// TIA Portal V20 export
FUNCTION_BLOCK "zPMC_Map"   // FB77, LAD
// stored: MemoryReserve 100, Namespace CITI_Logic, SetENOAutomatically false
   VAR_INPUT
      IN_AssistanceCall : Array[1..8] of Bool;
      IN_AssistanceCallAck : Array[1..8] of Bool;
      IN_Configuration : "CITI_Logic.zp_CITI_Configuration";
      IN_Data : "CITI_Logic.PMC_Input_Data";
   END_VAR
   VAR_OUTPUT
      OUT_Flasher_1Hz : Bool;   // 1Hz Flashing bit
      OUT_Team_Leader_Call_Out : Bool;   // ON when a Team Leader Call is active
      OUT_ShiftNumber : Byte;
   END_VAR
   VAR_IN_OUT
      PMC_Data : "CITI_Logic.zp_CITIData";
   END_VAR
   VAR
      MM_FaultWord_Zero : Bool;
      CycleTime_RUNNING_FB : Bool;   // Cycle Time Running set by this FB
      Cycle_END_OneShot_FB : Bool;   // Cycle End 1 Shot set by this FB
      System_Time_Tick : Time;   // System Time Tick
      Present_Time_Tick : Int;   // Present Time Tick
      Previous_Time_Tick : Int;   // Previous Time Tick
      Difference_Time_Tick : Int;   // Difference between Present and Previous Tick
      Difference_Time_DInt : DInt;   // Difference in Time
      CurrentProcessTime_DInt : DInt;   // Current Calculated Process Cycle Time
      CurrentPTimeConvertDInt : DInt;   // Current Process Cycle Time
      CurrentHeartBeatTim_DInt : DInt;   // Current Heartbeat Elapsed Time
      ShiftResetHold : Bool;   // Shift Hold Reset
      HeartBeatSetOneShot : Bool;   // Heartbeat Set 1 Shot
      DataReadySetup : Bool;   // Positive Edge of Data Ready
      CurrentLoadTime_DInt : DInt;   // Current Calculated Machine Load Cycle Time
      CurrentLTimeConvertDInt : DInt;   // Current Load Cycle Time
      CurrentUnLoadTime_DInt : DInt;   // Current Calculated Machine Unload Cycle Time
      CurrentUTimeConvertDInt : DInt;   // Current Unload Cycle Time
      CurrentPUNRdyDly_DInt : DInt;   // Current Pun Ready Delay Time
      TimerForDataReadySetup : DInt;   // Timer for Data Ready Setup1 Using Tick
      TimerForCycleTimeReady : DInt;   // Timer for Cycle Time Ready Using Tick
      TimerForFaultDelay : DInt;   // Timer for Fault Delay Using Tick
      Last_PUN_Data : String[20];
      FTQ_CurrDataRdyTime_DInt : DInt;   // Current Data Ready Time
      FTQ_Internal_Data_Ready : Bool;
      NullChar : Char;
      OneShotFirstScan : Bool;
      PUN_Is_NOT_Equal : Bool;
      PartType_NOT_Unknown : Bool;
      PartType_NOT_Equal : Bool;
      FaultStringIs9902 : Bool;
      TimerForFlasher : DInt;
      FB_OneShot : Array[1..32] of Bool;
   END_VAR
   VAR DB_SPECIFIC
      CurDTL { ExternalAccessible := 'False'; ExternalVisible := 'False'; ExternalWritable := 'False'} : DTL;   // Warning: Do not modify TEMP structure (affects clock synch)
      ON { ExternalAccessible := 'False'; ExternalVisible := 'False'; ExternalWritable := 'False'} : Bool;   // On
      OFF { ExternalAccessible := 'False'; ExternalVisible := 'False'; ExternalWritable := 'False'} : Bool;   // Off
      Temp_DINT { ExternalAccessible := 'False'; ExternalVisible := 'False'; ExternalWritable := 'False'} : DInt;   // Temporary Double Storage
      Temp_INT { ExternalAccessible := 'False'; ExternalVisible := 'False'; ExternalWritable := 'False'} : Int;   // Temporary Integer Storage
      Temp_LastCycle_Time { ExternalAccessible := 'False'; ExternalVisible := 'False'; ExternalWritable := 'False'} : DInt;   // Temporary to add the last load, process and unload times together into
      FTQ_t_ZERO { ExternalAccessible := 'False'; ExternalVisible := 'False'; ExternalWritable := 'False'} : Int;
   END_VAR
   VAR
      Fault_Load_Delay_Other_or_Unknown : IEC_TIMER;
      FlasherRatex2 { S7_SetPoint := 'True'} : DInt;
   END_VAR
   VAR_TEMP   // added for the SCL form of the ladder/FBD networks
      _w1 : Bool;
      _w2 : Bool;
      _w3 : Bool;
      _w4 : Bool;
      _w5 : Bool;
      _w6 : Bool;
      _w7 : Bool;
   END_VAR
BEGIN

REGION Network 1: Generate local "Always ON" and "Always OFF" conditions
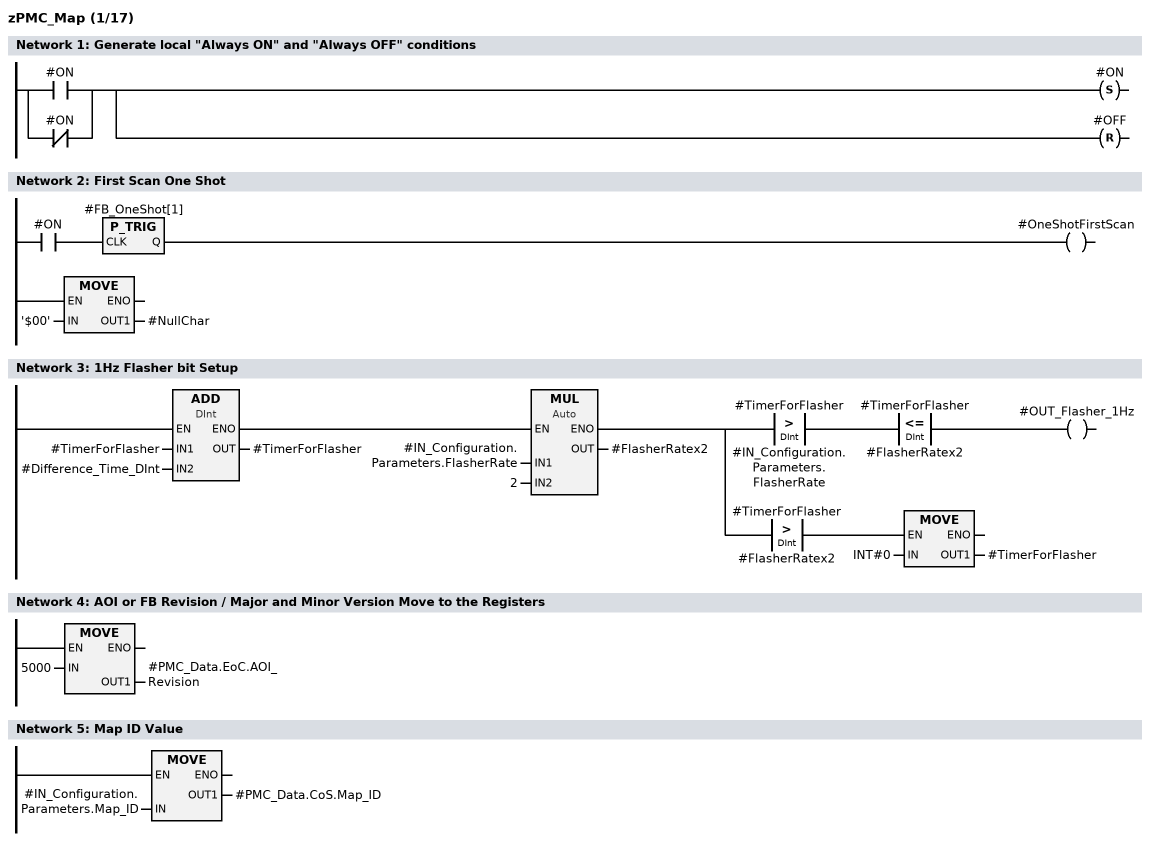
   RUNG wire#powerrail
      Contact( #ON )
      wire#w1
      S_Coil( #ON )
   END_RUNG
   RUNG wire#powerrail
      I_Contact( #ON )
   END_RUNG wire#w1
   RUNG wire#w1
      R_Coil( #OFF )
   END_RUNG
   // the same network as SCL:
   #_w1 := #ON OR NOT #ON;
   IF #_w1 THEN
       #ON := TRUE;
       #OFF := FALSE;
   END_IF;
END_REGION

REGION Network 2: First Scan One Shot
   RUNG wire#powerrail
      Contact( #ON )
      P_Trig( #FB_OneShot[1] )
      Coil( #OneShotFirstScan )
   END_RUNG
   RUNG wire#powerrail
      Move(in := '$00', out1 => #NullChar)
   END_RUNG
   // the same network as SCL:
   #_w1 := #ON AND NOT #FB_OneShot[1];   // rising edge
   #FB_OneShot[1] := #ON;
   #OneShotFirstScan := #_w1;
   #NullChar := '$00';
END_REGION

REGION Network 3: 1Hz Flasher bit Setup
   RUNG wire#powerrail
      { S7_Templates := "SrcType := DInt"; S7_GenerateENO := "TRUE" } Add(in1 := #TimerForFlasher, in2 := #Difference_Time_DInt, out => #TimerForFlasher)
      Mul(in1 := #IN_Configuration.Parameters.FlasherRate, in2 := 2, out => #FlasherRatex2)
      wire#w1
      { S7_Templates := "SrcType := DInt" } GT_Contact(in1 := #TimerForFlasher, in2 := #IN_Configuration.Parameters.FlasherRate)
      { S7_Templates := "SrcType := DInt" } LE_Contact(in1 := #TimerForFlasher, in2 := #FlasherRatex2)
      Coil( #OUT_Flasher_1Hz )
   END_RUNG
   RUNG wire#w1
      { S7_Templates := "SrcType := DInt" } GT_Contact(in1 := #TimerForFlasher, in2 := #FlasherRatex2)
      { S7_GenerateENO := "TRUE" } Move(in := INT#0, out1 => #TimerForFlasher)
   END_RUNG
   // the same network as SCL:
   // ENO of a box is taken as its EN; it also drops when the box reports an error
   #TimerForFlasher := #TimerForFlasher + #Difference_Time_DInt;
   #FlasherRatex2 := #IN_Configuration.Parameters.FlasherRate * 2;
   #OUT_Flasher_1Hz := (#TimerForFlasher > #IN_Configuration.Parameters.FlasherRate) AND (#TimerForFlasher <= #FlasherRatex2);
   IF #TimerForFlasher > #FlasherRatex2 THEN #TimerForFlasher := INT#0; END_IF;
END_REGION

REGION Network 4: AOI or FB Revision / Major and Minor Version Move to the Registers
   RUNG wire#powerrail
      { S7_GenerateENO := "TRUE" } Move(in := 5000, out1 => #PMC_Data.EoC.AOI_Revision)
   END_RUNG
   // the same network as SCL:
   #PMC_Data.EoC.AOI_Revision := 5000;
END_REGION

REGION Network 5: Map ID Value
   RUNG wire#powerrail
      Move(in := #IN_Configuration.Parameters.Map_ID, out1 => #PMC_Data.CoS.Map_ID)
   END_RUNG
   // the same network as SCL:
   #PMC_Data.CoS.Map_ID := #IN_Configuration.Parameters.Map_ID;
END_REGION

REGION Network 6: Assistance Calls and Acknowledge
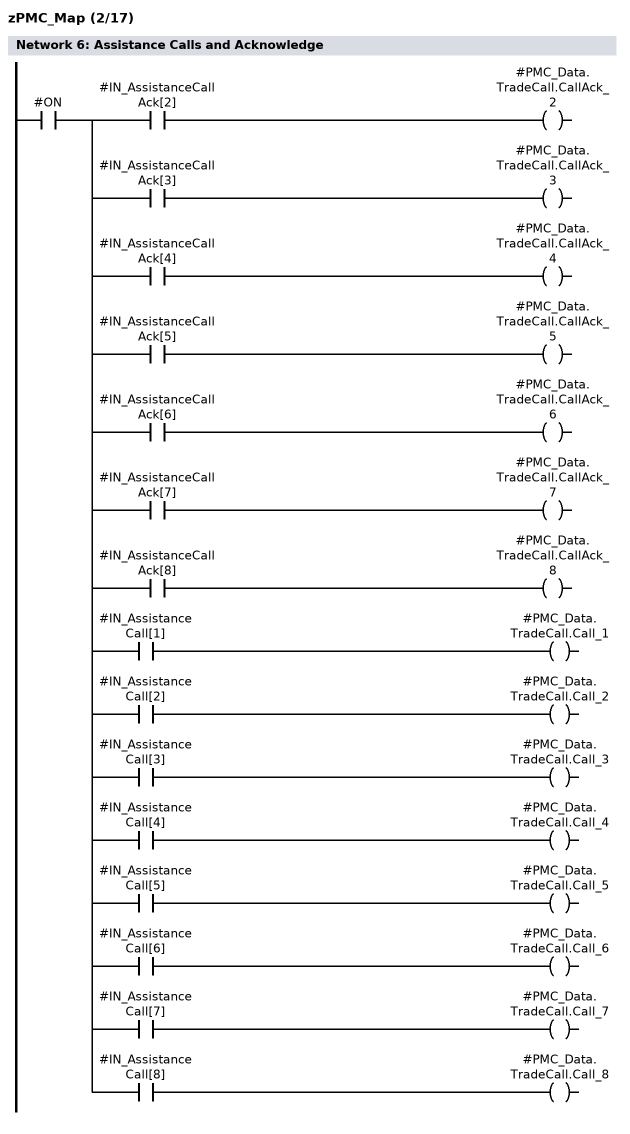
   RUNG wire#powerrail
      Contact( #ON )
      wire#w1
      Contact( #IN_AssistanceCallAck[2] )
      Coil( #PMC_Data.TradeCall.CallAck_2 )
   END_RUNG
   RUNG wire#w1
      Contact( #IN_AssistanceCallAck[3] )
      Coil( #PMC_Data.TradeCall.CallAck_3 )
   END_RUNG
   RUNG wire#w1
      Contact( #IN_AssistanceCallAck[4] )
      Coil( #PMC_Data.TradeCall.CallAck_4 )
   END_RUNG
   RUNG wire#w1
      Contact( #IN_AssistanceCallAck[5] )
      Coil( #PMC_Data.TradeCall.CallAck_5 )
   END_RUNG
   RUNG wire#w1
      Contact( #IN_AssistanceCallAck[6] )
      Coil( #PMC_Data.TradeCall.CallAck_6 )
   END_RUNG
   RUNG wire#w1
      Contact( #IN_AssistanceCallAck[7] )
      Coil( #PMC_Data.TradeCall.CallAck_7 )
   END_RUNG
   RUNG wire#w1
      Contact( #IN_AssistanceCallAck[8] )
      Coil( #PMC_Data.TradeCall.CallAck_8 )
   END_RUNG
   RUNG wire#w1
      Contact( #IN_AssistanceCall[1] )
      Coil( #PMC_Data.TradeCall.Call_1 )
   END_RUNG
   RUNG wire#w1
      Contact( #IN_AssistanceCall[2] )
      Coil( #PMC_Data.TradeCall.Call_2 )
   END_RUNG
   RUNG wire#w1
      Contact( #IN_AssistanceCall[3] )
      Coil( #PMC_Data.TradeCall.Call_3 )
   END_RUNG
   RUNG wire#w1
      Contact( #IN_AssistanceCall[4] )
      Coil( #PMC_Data.TradeCall.Call_4 )
   END_RUNG
   RUNG wire#w1
      Contact( #IN_AssistanceCall[5] )
      Coil( #PMC_Data.TradeCall.Call_5 )
   END_RUNG
   RUNG wire#w1
      Contact( #IN_AssistanceCall[6] )
      Coil( #PMC_Data.TradeCall.Call_6 )
   END_RUNG
   RUNG wire#w1
      Contact( #IN_AssistanceCall[7] )
      Coil( #PMC_Data.TradeCall.Call_7 )
   END_RUNG
   RUNG wire#w1
      Contact( #IN_AssistanceCall[8] )
      Coil( #PMC_Data.TradeCall.Call_8 )
   END_RUNG
   // the same network as SCL:
   #PMC_Data.TradeCall.CallAck_2 := #ON AND #IN_AssistanceCallAck[2];
   #PMC_Data.TradeCall.CallAck_3 := #ON AND #IN_AssistanceCallAck[3];
   #PMC_Data.TradeCall.CallAck_4 := #ON AND #IN_AssistanceCallAck[4];
   #PMC_Data.TradeCall.CallAck_5 := #ON AND #IN_AssistanceCallAck[5];
   #PMC_Data.TradeCall.CallAck_6 := #ON AND #IN_AssistanceCallAck[6];
   #PMC_Data.TradeCall.CallAck_7 := #ON AND #IN_AssistanceCallAck[7];
   #PMC_Data.TradeCall.CallAck_8 := #ON AND #IN_AssistanceCallAck[8];
   #PMC_Data.TradeCall.Call_1 := #ON AND #IN_AssistanceCall[1];
   #PMC_Data.TradeCall.Call_2 := #ON AND #IN_AssistanceCall[2];
   #PMC_Data.TradeCall.Call_3 := #ON AND #IN_AssistanceCall[3];
   #PMC_Data.TradeCall.Call_4 := #ON AND #IN_AssistanceCall[4];
   #PMC_Data.TradeCall.Call_5 := #ON AND #IN_AssistanceCall[5];
   #PMC_Data.TradeCall.Call_6 := #ON AND #IN_AssistanceCall[6];
   #PMC_Data.TradeCall.Call_7 := #ON AND #IN_AssistanceCall[7];
   #PMC_Data.TradeCall.Call_8 := #ON AND #IN_AssistanceCall[8];
END_REGION

REGION Network 7: Fault Word and Fault String Copy
   // This logic freezes the provided (changing) faultword from the input to this 
   // block.  This input should have been populated by template logic that has been 
   // appropriately modified as detailed in the Fault Logic procedure.
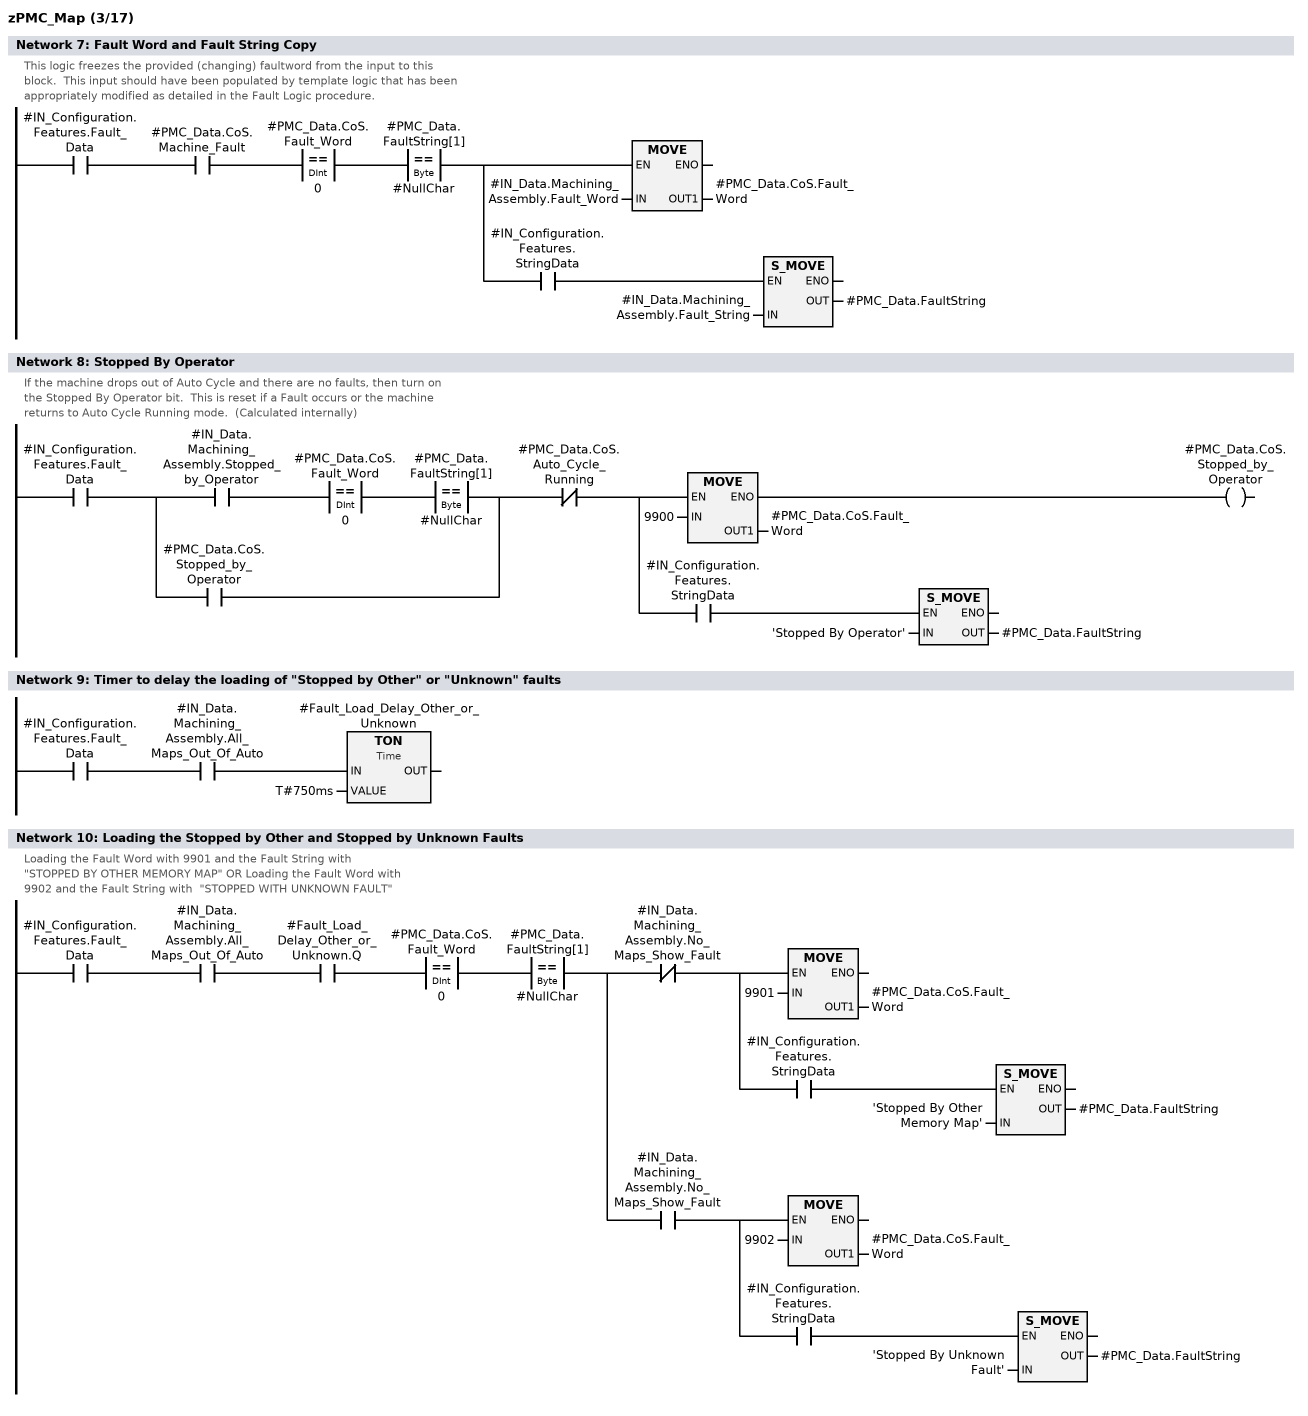
   RUNG wire#powerrail
      Contact( #IN_Configuration.Features.Fault_Data )
      Contact( #PMC_Data.CoS.Machine_Fault )
      { S7_Templates := "SrcType := DInt" } EQ_Contact(in1 := #PMC_Data.CoS.Fault_Word, in2 := 0)
      { S7_Templates := "SrcType := Byte" } EQ_Contact(in1 := #PMC_Data.FaultString[1], in2 := #NullChar)
      wire#w1
      { S7_GenerateENO := "TRUE" } Move(in := #IN_Data.Machining_Assembly.Fault_Word, out1 => #PMC_Data.CoS.Fault_Word)
   END_RUNG
   RUNG wire#w1
      Contact( #IN_Configuration.Features.StringData )
      S_Move(in := #IN_Data.Machining_Assembly.Fault_String, out => #PMC_Data.FaultString)
   END_RUNG
   // the same network as SCL:
   #_w1 := #IN_Configuration.Features.Fault_Data AND #PMC_Data.CoS.Machine_Fault AND (#PMC_Data.CoS.Fault_Word = 0) AND (#PMC_Data.FaultString[1] = #NullChar);
   IF #_w1 THEN #PMC_Data.CoS.Fault_Word := #IN_Data.Machining_Assembly.Fault_Word; END_IF;
   IF #_w1 AND #IN_Configuration.Features.StringData THEN
       #PMC_Data.FaultString := #IN_Data.Machining_Assembly.Fault_String;
   END_IF;
END_REGION

REGION Network 8: Stopped By Operator
   // If the machine drops out of Auto Cycle and there are no faults, then turn on 
   // the Stopped By Operator bit.  This is reset if a Fault occurs or the machine 
   // returns to Auto Cycle Running mode.  (Calculated internally)
   RUNG wire#powerrail
      Contact( #IN_Configuration.Features.Fault_Data )
      wire#w1
      Contact( #IN_Data.Machining_Assembly.Stopped_by_Operator )
      { S7_Templates := "SrcType := DInt" } EQ_Contact(in1 := #PMC_Data.CoS.Fault_Word, in2 := 0)
      { S7_Templates := "SrcType := Byte" } EQ_Contact(in1 := #PMC_Data.FaultString[1], in2 := #NullChar)
      wire#w2
      I_Contact( #PMC_Data.CoS.Auto_Cycle_Running )
      wire#w3
      { S7_GenerateENO := "TRUE" } Move(in := 9900, out1 => #PMC_Data.CoS.Fault_Word)
      Coil( #PMC_Data.CoS.Stopped_by_Operator )
   END_RUNG
   RUNG wire#w1
      Contact( #PMC_Data.CoS.Stopped_by_Operator )
   END_RUNG wire#w2
   RUNG wire#w3
      Contact( #IN_Configuration.Features.StringData )
      S_Move(in := 'Stopped By Operator', out => #PMC_Data.FaultString)
   END_RUNG
   // the same network as SCL:
   // ENO of a box is taken as its EN; it also drops when the box reports an error
   #_w1 := #IN_Configuration.Features.Fault_Data AND ((#IN_Data.Machining_Assembly.Stopped_by_Operator AND (#PMC_Data.CoS.Fault_Word = 0) AND (#PMC_Data.FaultString[1] = #NullChar)) OR #PMC_Data.CoS.Stopped_by_Operator) AND NOT #PMC_Data.CoS.Auto_Cycle_Running;
   IF #_w1 THEN #PMC_Data.CoS.Fault_Word := 9900; END_IF;
   #PMC_Data.CoS.Stopped_by_Operator := #_w1;
   IF #_w1 AND #IN_Configuration.Features.StringData THEN
       #PMC_Data.FaultString := 'Stopped By Operator';
   END_IF;
END_REGION

REGION Network 9: Timer to delay the loading of "Stopped by Other" or "Unknown" faults
   #Fault_Load_Delay_Other_or_Unknown.TON(IN := #IN_Configuration.Features.Fault_Data AND #IN_Data.Machining_Assembly.All_Maps_Out_Of_Auto, PT := T#750ms);   // TON coil
END_REGION

REGION Network 10: Loading the Stopped by Other and Stopped by Unknown Faults
   // Loading the Fault Word with 9901 and the Fault String with
   //  "STOPPED BY OTHER MEMORY MAP" OR Loading the Fault Word with 
   // 9902 and the Fault String with  "STOPPED WITH UNKNOWN FAULT"
   RUNG wire#powerrail
      Contact( #IN_Configuration.Features.Fault_Data )
      Contact( #IN_Data.Machining_Assembly.All_Maps_Out_Of_Auto )
      Contact( #Fault_Load_Delay_Other_or_Unknown.Q )
      { S7_Templates := "SrcType := DInt" } EQ_Contact(in1 := #PMC_Data.CoS.Fault_Word, in2 := 0)
      { S7_Templates := "SrcType := Byte" } EQ_Contact(in1 := #PMC_Data.FaultString[1], in2 := #NullChar)
      wire#w1
      I_Contact( #IN_Data.Machining_Assembly.No_Maps_Show_Fault )
      wire#w2
      { S7_GenerateENO := "TRUE" } Move(in := 9901, out1 => #PMC_Data.CoS.Fault_Word)
   END_RUNG
   RUNG wire#w2
      Contact( #IN_Configuration.Features.StringData )
      S_Move(in := 'Stopped By Other Memory Map', out => #PMC_Data.FaultString)
   END_RUNG
   RUNG wire#w1
      Contact( #IN_Data.Machining_Assembly.No_Maps_Show_Fault )
      wire#w3
      { S7_GenerateENO := "TRUE" } Move(in := 9902, out1 => #PMC_Data.CoS.Fault_Word)
   END_RUNG
   RUNG wire#w3
      Contact( #IN_Configuration.Features.StringData )
      S_Move(in := 'Stopped By Unknown Fault', out => #PMC_Data.FaultString)
   END_RUNG
   // the same network as SCL:
   #_w1 := #IN_Configuration.Features.Fault_Data AND #IN_Data.Machining_Assembly.All_Maps_Out_Of_Auto AND #Fault_Load_Delay_Other_or_Unknown.Q AND (#PMC_Data.CoS.Fault_Word = 0) AND (#PMC_Data.FaultString[1] = #NullChar);
   #_w2 := #_w1 AND NOT #IN_Data.Machining_Assembly.No_Maps_Show_Fault;
   IF #_w2 THEN #PMC_Data.CoS.Fault_Word := 9901; END_IF;
   IF #_w2 AND #IN_Configuration.Features.StringData THEN
       #PMC_Data.FaultString := 'Stopped By Other Memory Map';
   END_IF;
   #_w3 := #_w1 AND #IN_Data.Machining_Assembly.No_Maps_Show_Fault;
   IF #_w3 THEN #PMC_Data.CoS.Fault_Word := 9902; END_IF;
   IF #_w3 AND #IN_Configuration.Features.StringData THEN
       #PMC_Data.FaultString := 'Stopped By Unknown Fault';
   END_IF;
END_REGION

REGION Network 11: Sets a Bit for checking to see if the Fault String is 9902
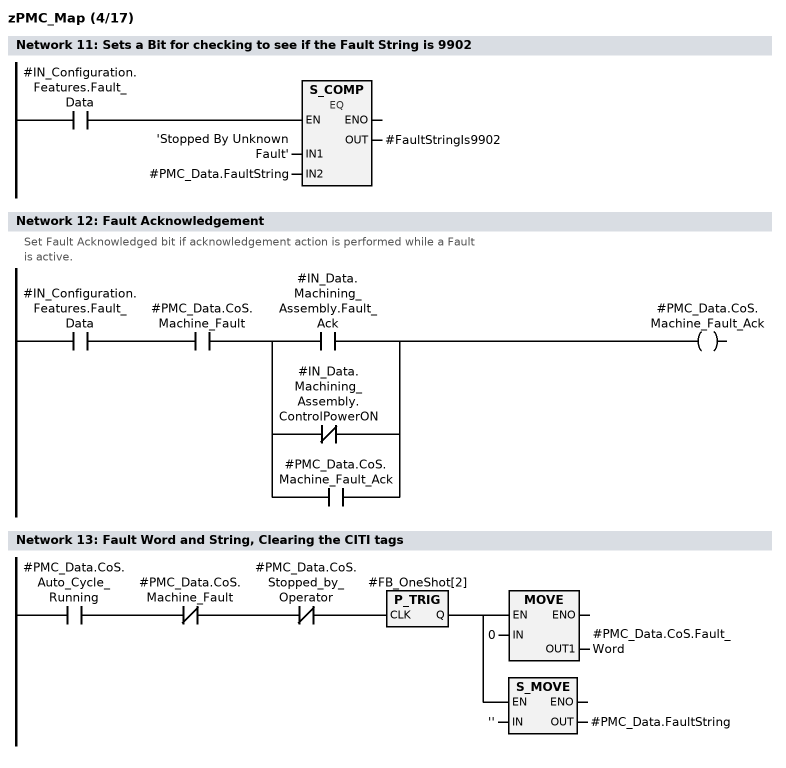
   RUNG wire#powerrail
      Contact( #IN_Configuration.Features.Fault_Data )
      { S7_Templates := "[relation := EQ, src_type := String]" } S_COMP(IN1 := 'Stopped By Unknown Fault', IN2 := #PMC_Data.FaultString, OUT => #FaultStringIs9902)
   END_RUNG
   // the same network as SCL:
   IF #IN_Configuration.Features.Fault_Data THEN
       S_COMP(IN1 := 'Stopped By Unknown Fault', IN2 := #PMC_Data.FaultString, OUT => #FaultStringIs9902);
   END_IF;
END_REGION

REGION Network 12: Fault Acknowledgement
   // Set Fault Acknowledged bit if acknowledgement action is performed while a Fault 
   // is active.
   RUNG wire#powerrail
      Contact( #IN_Configuration.Features.Fault_Data )
      Contact( #PMC_Data.CoS.Machine_Fault )
      wire#w1
      Contact( #IN_Data.Machining_Assembly.Fault_Ack )
      wire#w2
      Coil( #PMC_Data.CoS.Machine_Fault_Ack )
   END_RUNG
   RUNG wire#w1
      I_Contact( #IN_Data.Machining_Assembly.ControlPowerON )
   END_RUNG wire#w2
   RUNG wire#w1
      Contact( #PMC_Data.CoS.Machine_Fault_Ack )
   END_RUNG wire#w2
   // the same network as SCL:
   #PMC_Data.CoS.Machine_Fault_Ack := #IN_Configuration.Features.Fault_Data AND #PMC_Data.CoS.Machine_Fault AND (#IN_Data.Machining_Assembly.Fault_Ack OR NOT #IN_Data.Machining_Assembly.ControlPowerON OR #PMC_Data.CoS.Machine_Fault_Ack);
END_REGION

REGION Network 13: Fault Word and String, Clearing the CITI tags
   RUNG wire#powerrail
      Contact( #PMC_Data.CoS.Auto_Cycle_Running )
      I_Contact( #PMC_Data.CoS.Machine_Fault )
      I_Contact( #PMC_Data.CoS.Stopped_by_Operator )
      P_Trig( #FB_OneShot[2] )
      wire#w1
      { S7_GenerateENO := "TRUE" } Move(in := 0, out1 => #PMC_Data.CoS.Fault_Word)
   END_RUNG
   RUNG wire#w1
      S_Move(in := '', out => #PMC_Data.FaultString)
   END_RUNG
   // the same network as SCL:
   #_w1 := #PMC_Data.CoS.Auto_Cycle_Running AND NOT #PMC_Data.CoS.Machine_Fault AND NOT #PMC_Data.CoS.Stopped_by_Operator;
   #_w2 := #_w1 AND NOT #FB_OneShot[2];   // rising edge
   #FB_OneShot[2] := #_w1;
   IF #_w2 THEN
       #PMC_Data.CoS.Fault_Word := 0;
       #PMC_Data.FaultString := '';
   END_IF;
END_REGION

REGION Network 14: Copy Boolean Data into DB / Copy Interface Data into DB
   // For inputs that are already determined, or that can be easily determined, they 
   // are calculated and/or copied directly into the Memory Map DB so that they are 
   // available for the remainder of the FB.
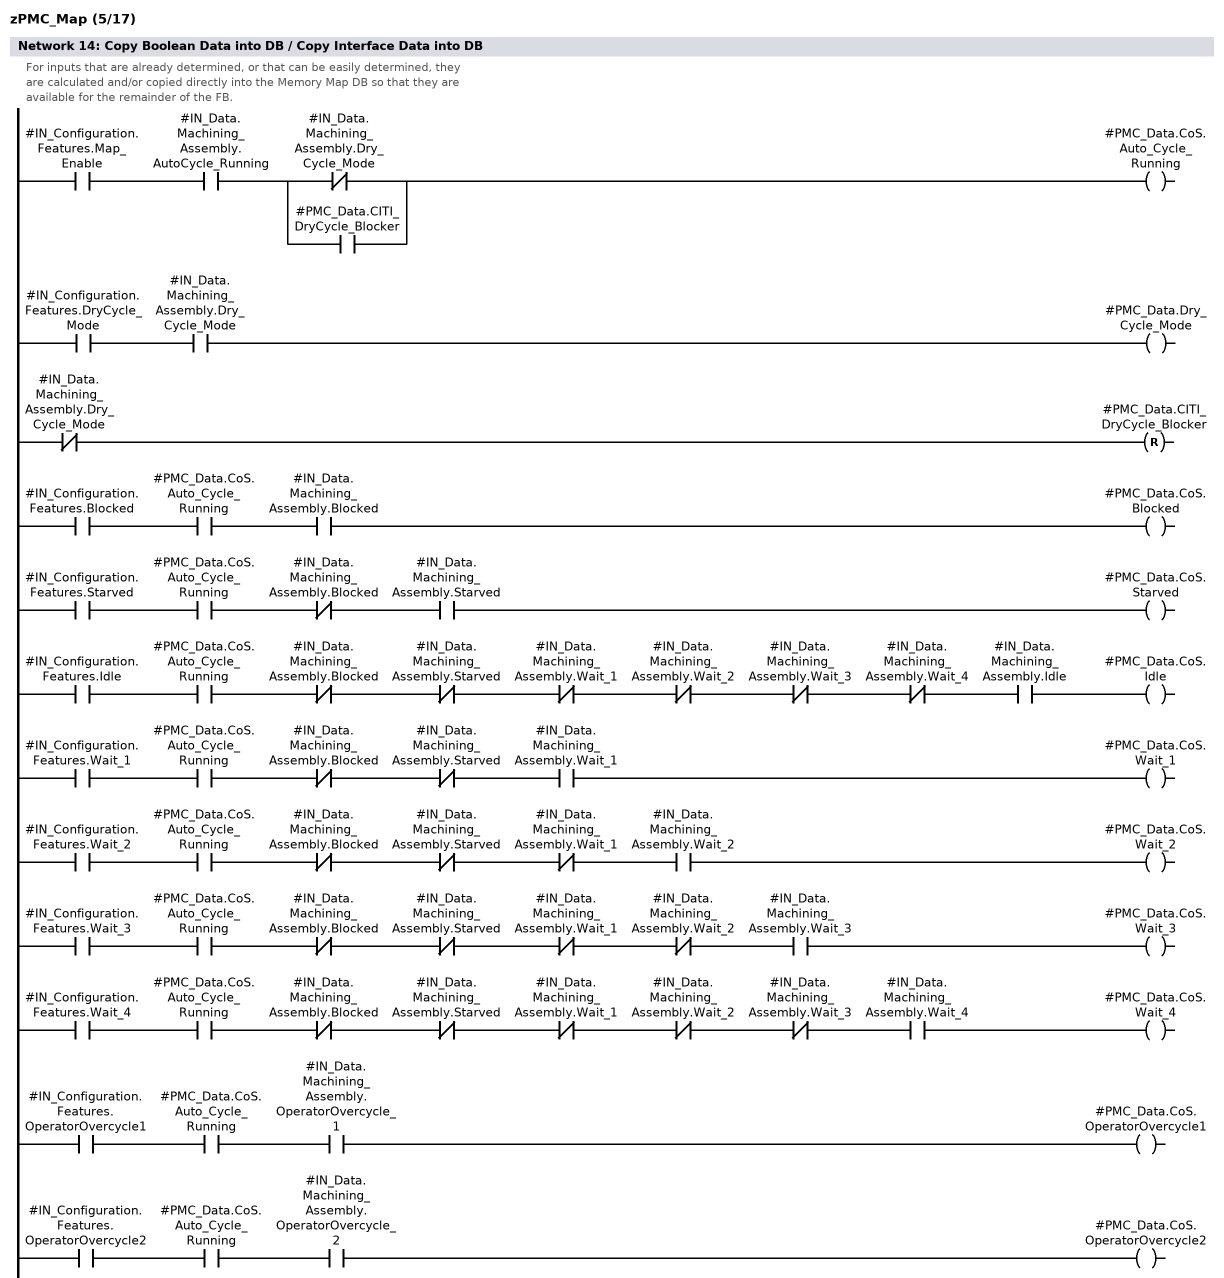
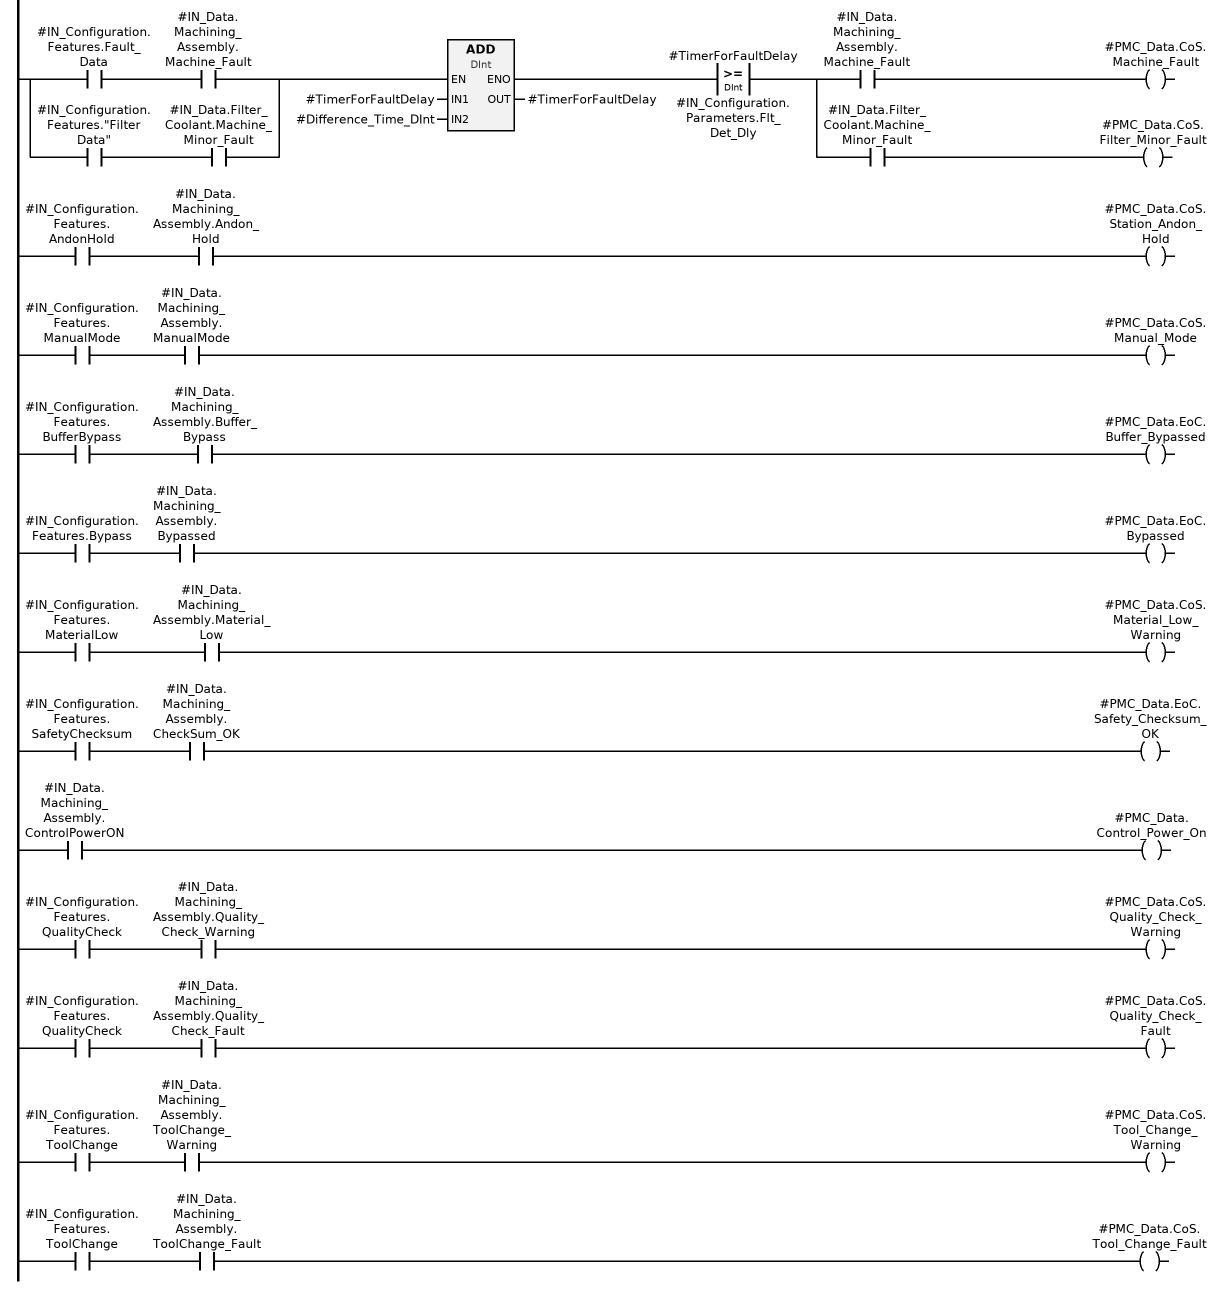
   RUNG wire#powerrail
      Contact( #IN_Configuration.Features.Map_Enable )
      Contact( #IN_Data.Machining_Assembly.AutoCycle_Running )
      wire#w1
      I_Contact( #IN_Data.Machining_Assembly.Dry_Cycle_Mode )
      wire#w2
      Coil( #PMC_Data.CoS.Auto_Cycle_Running )
   END_RUNG
   RUNG wire#w1
      Contact( #PMC_Data.CITI_DryCycle_Blocker )
   END_RUNG wire#w2
   RUNG wire#powerrail
      Contact( #IN_Configuration.Features.DryCycle_Mode )
      Contact( #IN_Data.Machining_Assembly.Dry_Cycle_Mode )
      Coil( #PMC_Data.Dry_Cycle_Mode )
   END_RUNG
   RUNG wire#powerrail
      I_Contact( #IN_Data.Machining_Assembly.Dry_Cycle_Mode )
      R_Coil( #PMC_Data.CITI_DryCycle_Blocker )
   END_RUNG
   RUNG wire#powerrail
      Contact( #IN_Configuration.Features.Blocked )
      Contact( #PMC_Data.CoS.Auto_Cycle_Running )
      Contact( #IN_Data.Machining_Assembly.Blocked )
      Coil( #PMC_Data.CoS.Blocked )
   END_RUNG
   RUNG wire#powerrail
      Contact( #IN_Configuration.Features.Starved )
      Contact( #PMC_Data.CoS.Auto_Cycle_Running )
      I_Contact( #IN_Data.Machining_Assembly.Blocked )
      Contact( #IN_Data.Machining_Assembly.Starved )
      Coil( #PMC_Data.CoS.Starved )
   END_RUNG
   RUNG wire#powerrail
      Contact( #IN_Configuration.Features.Idle )
      Contact( #PMC_Data.CoS.Auto_Cycle_Running )
      I_Contact( #IN_Data.Machining_Assembly.Blocked )
      I_Contact( #IN_Data.Machining_Assembly.Starved )
      I_Contact( #IN_Data.Machining_Assembly.Wait_1 )
      I_Contact( #IN_Data.Machining_Assembly.Wait_2 )
      I_Contact( #IN_Data.Machining_Assembly.Wait_3 )
      I_Contact( #IN_Data.Machining_Assembly.Wait_4 )
      Contact( #IN_Data.Machining_Assembly.Idle )
      Coil( #PMC_Data.CoS.Idle )
   END_RUNG
   RUNG wire#powerrail
      Contact( #IN_Configuration.Features.Wait_1 )
      Contact( #PMC_Data.CoS.Auto_Cycle_Running )
      I_Contact( #IN_Data.Machining_Assembly.Blocked )
      I_Contact( #IN_Data.Machining_Assembly.Starved )
      Contact( #IN_Data.Machining_Assembly.Wait_1 )
      Coil( #PMC_Data.CoS.Wait_1 )
   END_RUNG
   RUNG wire#powerrail
      Contact( #IN_Configuration.Features.Wait_2 )
      Contact( #PMC_Data.CoS.Auto_Cycle_Running )
      I_Contact( #IN_Data.Machining_Assembly.Blocked )
      I_Contact( #IN_Data.Machining_Assembly.Starved )
      I_Contact( #IN_Data.Machining_Assembly.Wait_1 )
      Contact( #IN_Data.Machining_Assembly.Wait_2 )
      Coil( #PMC_Data.CoS.Wait_2 )
   END_RUNG
   RUNG wire#powerrail
      Contact( #IN_Configuration.Features.Wait_3 )
      Contact( #PMC_Data.CoS.Auto_Cycle_Running )
      I_Contact( #IN_Data.Machining_Assembly.Blocked )
      I_Contact( #IN_Data.Machining_Assembly.Starved )
      I_Contact( #IN_Data.Machining_Assembly.Wait_1 )
      I_Contact( #IN_Data.Machining_Assembly.Wait_2 )
      Contact( #IN_Data.Machining_Assembly.Wait_3 )
      Coil( #PMC_Data.CoS.Wait_3 )
   END_RUNG
   RUNG wire#powerrail
      Contact( #IN_Configuration.Features.Wait_4 )
      Contact( #PMC_Data.CoS.Auto_Cycle_Running )
      I_Contact( #IN_Data.Machining_Assembly.Blocked )
      I_Contact( #IN_Data.Machining_Assembly.Starved )
      I_Contact( #IN_Data.Machining_Assembly.Wait_1 )
      I_Contact( #IN_Data.Machining_Assembly.Wait_2 )
      I_Contact( #IN_Data.Machining_Assembly.Wait_3 )
      Contact( #IN_Data.Machining_Assembly.Wait_4 )
      Coil( #PMC_Data.CoS.Wait_4 )
   END_RUNG
   RUNG wire#powerrail
      Contact( #IN_Configuration.Features.OperatorOvercycle1 )
      Contact( #PMC_Data.CoS.Auto_Cycle_Running )
      Contact( #IN_Data.Machining_Assembly.OperatorOvercycle_1 )
      Coil( #PMC_Data.CoS.OperatorOvercycle1 )
   END_RUNG
   RUNG wire#powerrail
      Contact( #IN_Configuration.Features.OperatorOvercycle2 )
      Contact( #PMC_Data.CoS.Auto_Cycle_Running )
      Contact( #IN_Data.Machining_Assembly.OperatorOvercycle_2 )
      Coil( #PMC_Data.CoS.OperatorOvercycle2 )
   END_RUNG
   RUNG wire#powerrail
      Contact( #IN_Configuration.Features.Fault_Data )
      Contact( #IN_Data.Machining_Assembly.Machine_Fault )
      wire#w3
      { S7_Templates := "SrcType := DInt" } Add(in1 := #TimerForFaultDelay, in2 := #Difference_Time_DInt, out => #TimerForFaultDelay)
      { S7_Templates := "SrcType := DInt" } GE_Contact(in1 := #TimerForFaultDelay, in2 := #IN_Configuration.Parameters.Flt_Det_Dly)
      wire#w4
      Contact( #IN_Data.Machining_Assembly.Machine_Fault )
      Coil( #PMC_Data.CoS.Machine_Fault )
   END_RUNG
   RUNG wire#powerrail
      Contact( #IN_Configuration.Features."Filter Data" )
      Contact( #IN_Data.Filter_Coolant.Machine_Minor_Fault )
   END_RUNG wire#w3
   RUNG wire#w4
      Contact( #IN_Data.Filter_Coolant.Machine_Minor_Fault )
      Coil( #PMC_Data.CoS.Filter_Minor_Fault )
   END_RUNG
   RUNG wire#powerrail
      Contact( #IN_Configuration.Features.AndonHold )
      Contact( #IN_Data.Machining_Assembly.Andon_Hold )
      Coil( #PMC_Data.CoS.Station_Andon_Hold )
   END_RUNG
   RUNG wire#powerrail
      Contact( #IN_Configuration.Features.ManualMode )
      Contact( #IN_Data.Machining_Assembly.ManualMode )
      Coil( #PMC_Data.CoS.Manual_Mode )
   END_RUNG
   RUNG wire#powerrail
      Contact( #IN_Configuration.Features.BufferBypass )
      Contact( #IN_Data.Machining_Assembly.Buffer_Bypass )
      Coil( #PMC_Data.EoC.Buffer_Bypassed )
   END_RUNG
   RUNG wire#powerrail
      Contact( #IN_Configuration.Features.Bypass )
      Contact( #IN_Data.Machining_Assembly.Bypassed )
      Coil( #PMC_Data.EoC.Bypassed )
   END_RUNG
   RUNG wire#powerrail
      Contact( #IN_Configuration.Features.MaterialLow )
      Contact( #IN_Data.Machining_Assembly.Material_Low )
      Coil( #PMC_Data.CoS.Material_Low_Warning )
   END_RUNG
   RUNG wire#powerrail
      Contact( #IN_Configuration.Features.SafetyChecksum )
      Contact( #IN_Data.Machining_Assembly.CheckSum_OK )
      Coil( #PMC_Data.EoC.Safety_Checksum_OK )
   END_RUNG
   RUNG wire#powerrail
      Contact( #IN_Data.Machining_Assembly.ControlPowerON )
      Coil( #PMC_Data.Control_Power_On )
   END_RUNG
   RUNG wire#powerrail
      Contact( #IN_Configuration.Features.QualityCheck )
      Contact( #IN_Data.Machining_Assembly.Quality_Check_Warning )
      Coil( #PMC_Data.CoS.Quality_Check_Warning )
   END_RUNG
   RUNG wire#powerrail
      Contact( #IN_Configuration.Features.QualityCheck )
      Contact( #IN_Data.Machining_Assembly.Quality_Check_Fault )
      Coil( #PMC_Data.CoS.Quality_Check_Fault )
   END_RUNG
   RUNG wire#powerrail
      Contact( #IN_Configuration.Features.ToolChange )
      Contact( #IN_Data.Machining_Assembly.ToolChange_Warning )
      Coil( #PMC_Data.CoS.Tool_Change_Warning )
   END_RUNG
   RUNG wire#powerrail
      Contact( #IN_Configuration.Features.ToolChange )
      Contact( #IN_Data.Machining_Assembly.ToolChange_Fault )
      Coil( #PMC_Data.CoS.Tool_Change_Fault )
   END_RUNG
   // the same network as SCL:
   #PMC_Data.CoS.Auto_Cycle_Running := #IN_Configuration.Features.Map_Enable AND #IN_Data.Machining_Assembly.AutoCycle_Running AND (NOT #IN_Data.Machining_Assembly.Dry_Cycle_Mode OR #PMC_Data.CITI_DryCycle_Blocker);
   #PMC_Data.Dry_Cycle_Mode := #IN_Configuration.Features.DryCycle_Mode AND #IN_Data.Machining_Assembly.Dry_Cycle_Mode;
   IF NOT #IN_Data.Machining_Assembly.Dry_Cycle_Mode THEN #PMC_Data.CITI_DryCycle_Blocker := FALSE; END_IF;
   #PMC_Data.CoS.Blocked := #IN_Configuration.Features.Blocked AND #PMC_Data.CoS.Auto_Cycle_Running AND #IN_Data.Machining_Assembly.Blocked;
   #PMC_Data.CoS.Starved := #IN_Configuration.Features.Starved AND #PMC_Data.CoS.Auto_Cycle_Running AND NOT #IN_Data.Machining_Assembly.Blocked AND #IN_Data.Machining_Assembly.Starved;
   #PMC_Data.CoS.Idle := #IN_Configuration.Features.Idle AND #PMC_Data.CoS.Auto_Cycle_Running AND NOT #IN_Data.Machining_Assembly.Blocked AND NOT #IN_Data.Machining_Assembly.Starved AND NOT #IN_Data.Machining_Assembly.Wait_1 AND NOT #IN_Data.Machining_Assembly.Wait_2 AND NOT #IN_Data.Machining_Assembly.Wait_3 AND NOT #IN_Data.Machining_Assembly.Wait_4 AND #IN_Data.Machining_Assembly.Idle;
   #PMC_Data.CoS.Wait_1 := #IN_Configuration.Features.Wait_1 AND #PMC_Data.CoS.Auto_Cycle_Running AND NOT #IN_Data.Machining_Assembly.Blocked AND NOT #IN_Data.Machining_Assembly.Starved AND #IN_Data.Machining_Assembly.Wait_1;
   #PMC_Data.CoS.Wait_2 := #IN_Configuration.Features.Wait_2 AND #PMC_Data.CoS.Auto_Cycle_Running AND NOT #IN_Data.Machining_Assembly.Blocked AND NOT #IN_Data.Machining_Assembly.Starved AND NOT #IN_Data.Machining_Assembly.Wait_1 AND #IN_Data.Machining_Assembly.Wait_2;
   #PMC_Data.CoS.Wait_3 := #IN_Configuration.Features.Wait_3 AND #PMC_Data.CoS.Auto_Cycle_Running AND NOT #IN_Data.Machining_Assembly.Blocked AND NOT #IN_Data.Machining_Assembly.Starved AND NOT #IN_Data.Machining_Assembly.Wait_1 AND NOT #IN_Data.Machining_Assembly.Wait_2 AND #IN_Data.Machining_Assembly.Wait_3;
   #PMC_Data.CoS.Wait_4 := #IN_Configuration.Features.Wait_4 AND #PMC_Data.CoS.Auto_Cycle_Running AND NOT #IN_Data.Machining_Assembly.Blocked AND NOT #IN_Data.Machining_Assembly.Starved AND NOT #IN_Data.Machining_Assembly.Wait_1 AND NOT #IN_Data.Machining_Assembly.Wait_2 AND NOT #IN_Data.Machining_Assembly.Wait_3 AND #IN_Data.Machining_Assembly.Wait_4;
   #PMC_Data.CoS.OperatorOvercycle1 := #IN_Configuration.Features.OperatorOvercycle1 AND #PMC_Data.CoS.Auto_Cycle_Running AND #IN_Data.Machining_Assembly.OperatorOvercycle_1;
   #PMC_Data.CoS.OperatorOvercycle2 := #IN_Configuration.Features.OperatorOvercycle2 AND #PMC_Data.CoS.Auto_Cycle_Running AND #IN_Data.Machining_Assembly.OperatorOvercycle_2;
   #_w1 := (#IN_Configuration.Features.Fault_Data AND #IN_Data.Machining_Assembly.Machine_Fault) OR (#IN_Configuration.Features."Filter Data" AND #IN_Data.Filter_Coolant.Machine_Minor_Fault);
   IF #_w1 THEN #TimerForFaultDelay := #TimerForFaultDelay + #Difference_Time_DInt; END_IF;
   #_w2 := #_w1 AND (#TimerForFaultDelay >= #IN_Configuration.Parameters.Flt_Det_Dly);
   #PMC_Data.CoS.Machine_Fault := #_w2 AND #IN_Data.Machining_Assembly.Machine_Fault;
   #PMC_Data.CoS.Filter_Minor_Fault := #_w2 AND #IN_Data.Filter_Coolant.Machine_Minor_Fault;
   #PMC_Data.CoS.Station_Andon_Hold := #IN_Configuration.Features.AndonHold AND #IN_Data.Machining_Assembly.Andon_Hold;
   #PMC_Data.CoS.Manual_Mode := #IN_Configuration.Features.ManualMode AND #IN_Data.Machining_Assembly.ManualMode;
   #PMC_Data.EoC.Buffer_Bypassed := #IN_Configuration.Features.BufferBypass AND #IN_Data.Machining_Assembly.Buffer_Bypass;
   #PMC_Data.EoC.Bypassed := #IN_Configuration.Features.Bypass AND #IN_Data.Machining_Assembly.Bypassed;
   #PMC_Data.CoS.Material_Low_Warning := #IN_Configuration.Features.MaterialLow AND #IN_Data.Machining_Assembly.Material_Low;
   #PMC_Data.EoC.Safety_Checksum_OK := #IN_Configuration.Features.SafetyChecksum AND #IN_Data.Machining_Assembly.CheckSum_OK;
   #PMC_Data.Control_Power_On := #IN_Data.Machining_Assembly.ControlPowerON;
   #PMC_Data.CoS.Quality_Check_Warning := #IN_Configuration.Features.QualityCheck AND #IN_Data.Machining_Assembly.Quality_Check_Warning;
   #PMC_Data.CoS.Quality_Check_Fault := #IN_Configuration.Features.QualityCheck AND #IN_Data.Machining_Assembly.Quality_Check_Fault;
   #PMC_Data.CoS.Tool_Change_Warning := #IN_Configuration.Features.ToolChange AND #IN_Data.Machining_Assembly.ToolChange_Warning;
   #PMC_Data.CoS.Tool_Change_Fault := #IN_Configuration.Features.ToolChange AND #IN_Data.Machining_Assembly.ToolChange_Fault;
END_REGION

REGION Network 15: Part Type Data
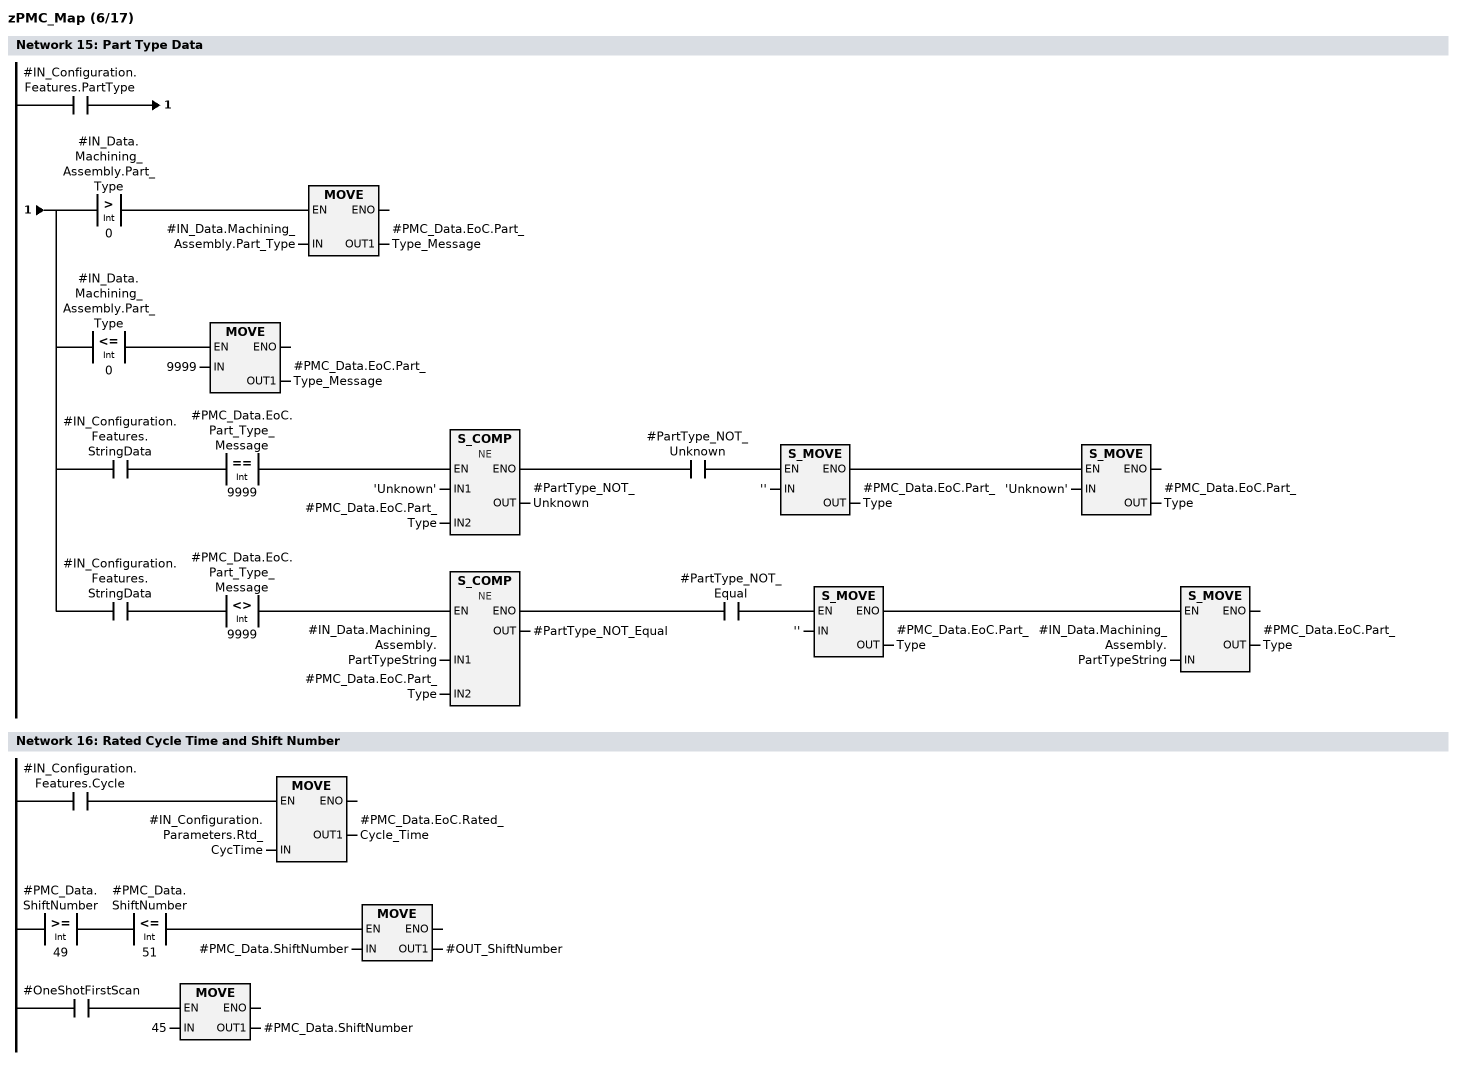
   RUNG wire#powerrail
      Contact( #IN_Configuration.Features.PartType )
      wire#w1
      { S7_Templates := "SrcType := Int" } GT_Contact(in1 := #IN_Data.Machining_Assembly.Part_Type, in2 := 0)
      Move(in := #IN_Data.Machining_Assembly.Part_Type, out1 => #PMC_Data.EoC.Part_Type_Message)
   END_RUNG
   RUNG wire#w1
      { S7_Templates := "SrcType := Int" } LE_Contact(in1 := #IN_Data.Machining_Assembly.Part_Type, in2 := 0)
      Move(in := 9999, out1 => #PMC_Data.EoC.Part_Type_Message)
   END_RUNG
   RUNG wire#w1
      Contact( #IN_Configuration.Features.StringData )
      { S7_Templates := "SrcType := Int" } EQ_Contact(in1 := #PMC_Data.EoC.Part_Type_Message, in2 := 9999)
      { S7_Templates := "[relation := NE, src_type := String]" } S_COMP(IN1 := 'Unknown', IN2 := #PMC_Data.EoC.Part_Type, OUT => #PartType_NOT_Unknown)
      Contact( #PartType_NOT_Unknown )
      S_Move(in := '', out => #PMC_Data.EoC.Part_Type)
      S_Move(in := 'Unknown', out => #PMC_Data.EoC.Part_Type)
   END_RUNG
   RUNG wire#w1
      Contact( #IN_Configuration.Features.StringData )
      { S7_Templates := "SrcType := Int" } NE_Contact(in1 := #PMC_Data.EoC.Part_Type_Message, in2 := 9999)
      { S7_Templates := "[relation := NE, src_type := String]" } S_COMP(IN1 := #IN_Data.Machining_Assembly.PartTypeString, IN2 := #PMC_Data.EoC.Part_Type, OUT => #PartType_NOT_Equal)
      Contact( #PartType_NOT_Equal )
      S_Move(in := '', out => #PMC_Data.EoC.Part_Type)
      S_Move(in := #IN_Data.Machining_Assembly.PartTypeString, out => #PMC_Data.EoC.Part_Type)
   END_RUNG
   // the same network as SCL:
   IF #IN_Configuration.Features.PartType AND (#IN_Data.Machining_Assembly.Part_Type > 0) THEN
       #PMC_Data.EoC.Part_Type_Message := #IN_Data.Machining_Assembly.Part_Type;
   END_IF;
   IF #IN_Configuration.Features.PartType AND (#IN_Data.Machining_Assembly.Part_Type <= 0) THEN
       #PMC_Data.EoC.Part_Type_Message := 9999;
   END_IF;
   #_w1 := #IN_Configuration.Features.PartType AND #IN_Configuration.Features.StringData AND (#PMC_Data.EoC.Part_Type_Message = 9999);
   S_COMP(EN := #_w1,
          IN1 := 'Unknown',
          IN2 := #PMC_Data.EoC.Part_Type,
          OUT => #PartType_NOT_Unknown,
          ENO => #_w2);
   IF #_w2 AND #PartType_NOT_Unknown THEN
       #PMC_Data.EoC.Part_Type := '';
       #PMC_Data.EoC.Part_Type := 'Unknown';
   END_IF;
   #_w3 := #IN_Configuration.Features.PartType AND #IN_Configuration.Features.StringData AND (#PMC_Data.EoC.Part_Type_Message <> 9999);
   S_COMP(EN := #_w3,
          IN1 := #IN_Data.Machining_Assembly.PartTypeString,
          IN2 := #PMC_Data.EoC.Part_Type,
          OUT => #PartType_NOT_Equal,
          ENO => #_w4);
   IF #_w4 AND #PartType_NOT_Equal THEN
       #PMC_Data.EoC.Part_Type := '';
       #PMC_Data.EoC.Part_Type := #IN_Data.Machining_Assembly.PartTypeString;
   END_IF;
END_REGION

REGION Network 16: Rated Cycle Time and Shift Number
   RUNG wire#powerrail
      Contact( #IN_Configuration.Features.Cycle )
      Move(in := #IN_Configuration.Parameters.Rtd_CycTime, out1 => #PMC_Data.EoC.Rated_Cycle_Time)
   END_RUNG
   RUNG wire#powerrail
      { S7_Templates := "SrcType := Int" } GE_Contact(in1 := #PMC_Data.ShiftNumber, in2 := 49)
      { S7_Templates := "SrcType := Int" } LE_Contact(in1 := #PMC_Data.ShiftNumber, in2 := 51)
      Move(in := #PMC_Data.ShiftNumber, out1 => #OUT_ShiftNumber)
   END_RUNG
   RUNG wire#powerrail
      Contact( #OneShotFirstScan )
      Move(in := 45, out1 => #PMC_Data.ShiftNumber)
   END_RUNG
   // the same network as SCL:
   IF #IN_Configuration.Features.Cycle THEN
       #PMC_Data.EoC.Rated_Cycle_Time := #IN_Configuration.Parameters.Rtd_CycTime;
   END_IF;
   IF (#PMC_Data.ShiftNumber >= 49) AND (#PMC_Data.ShiftNumber <= 51) THEN
       #OUT_ShiftNumber := #PMC_Data.ShiftNumber;
   END_IF;
   IF #OneShotFirstScan THEN #PMC_Data.ShiftNumber := 45; END_IF;
END_REGION

REGION Network 17: PUN / GM Part Number / Optional Data
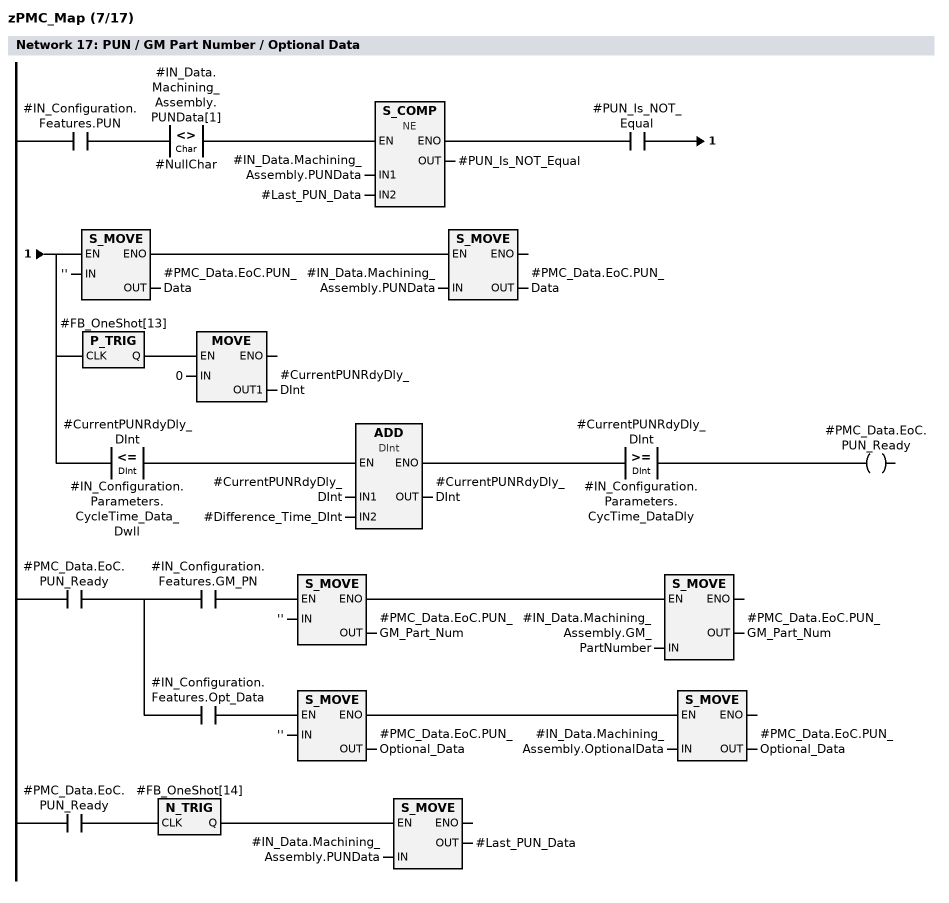
   RUNG wire#powerrail
      Contact( #IN_Configuration.Features.PUN )
      { S7_Templates := "SrcType := Char" } NE_Contact(in1 := #IN_Data.Machining_Assembly.PUNData[1], in2 := #NullChar)
      { S7_Templates := "[relation := NE, src_type := String]" } S_COMP(IN1 := #IN_Data.Machining_Assembly.PUNData, IN2 := #Last_PUN_Data, OUT => #PUN_Is_NOT_Equal)
      Contact( #PUN_Is_NOT_Equal )
      wire#w1
      S_Move(in := '', out => #PMC_Data.EoC.PUN_Data)
      S_Move(in := #IN_Data.Machining_Assembly.PUNData, out => #PMC_Data.EoC.PUN_Data)
   END_RUNG
   RUNG wire#w1
      P_Trig( #FB_OneShot[13] )
      Move(in := 0, out1 => #CurrentPUNRdyDly_DInt)
   END_RUNG
   RUNG wire#w1
      { S7_Templates := "SrcType := DInt" } LE_Contact(in1 := #CurrentPUNRdyDly_DInt, in2 := #IN_Configuration.Parameters.CycleTime_Data_Dwll)
      { S7_Templates := "SrcType := DInt" } Add(in1 := #CurrentPUNRdyDly_DInt, in2 := #Difference_Time_DInt, out => #CurrentPUNRdyDly_DInt)
      { S7_Templates := "SrcType := DInt" } GE_Contact(in1 := #CurrentPUNRdyDly_DInt, in2 := #IN_Configuration.Parameters.CycTime_DataDly)
      Coil( #PMC_Data.EoC.PUN_Ready )
   END_RUNG
   RUNG wire#powerrail
      Contact( #PMC_Data.EoC.PUN_Ready )
      wire#w2
      Contact( #IN_Configuration.Features.GM_PN )
      S_Move(in := '', out => #PMC_Data.EoC.PUN_GM_Part_Num)
      S_Move(in := #IN_Data.Machining_Assembly.GM_PartNumber, out => #PMC_Data.EoC.PUN_GM_Part_Num)
   END_RUNG
   RUNG wire#w2
      Contact( #IN_Configuration.Features.Opt_Data )
      S_Move(in := '', out => #PMC_Data.EoC.PUN_Optional_Data)
      S_Move(in := #IN_Data.Machining_Assembly.OptionalData, out => #PMC_Data.EoC.PUN_Optional_Data)
   END_RUNG
   RUNG wire#powerrail
      Contact( #PMC_Data.EoC.PUN_Ready )
      N_Trig( #FB_OneShot[14] )
      S_Move(in := #IN_Data.Machining_Assembly.PUNData, out => #Last_PUN_Data)
   END_RUNG
   // the same network as SCL:
   #_w1 := #IN_Configuration.Features.PUN AND (#IN_Data.Machining_Assembly.PUNData[1] <> #NullChar);
   S_COMP(EN := #_w1,
          IN1 := #IN_Data.Machining_Assembly.PUNData,
          IN2 := #Last_PUN_Data,
          OUT => #PUN_Is_NOT_Equal,
          ENO => #_w2);
   #_w3 := #_w2 AND #PUN_Is_NOT_Equal;
   IF #_w3 THEN
       #PMC_Data.EoC.PUN_Data := '';
       #PMC_Data.EoC.PUN_Data := #IN_Data.Machining_Assembly.PUNData;
   END_IF;
   #_w4 := #_w3 AND NOT #FB_OneShot[13];   // rising edge
   #FB_OneShot[13] := #_w3;
   IF #_w4 THEN #CurrentPUNRdyDly_DInt := 0; END_IF;
   #_w5 := #_w3 AND (#CurrentPUNRdyDly_DInt <= #IN_Configuration.Parameters.CycleTime_Data_Dwll);
   IF #_w5 THEN #CurrentPUNRdyDly_DInt := #CurrentPUNRdyDly_DInt + #Difference_Time_DInt; END_IF;
   #PMC_Data.EoC.PUN_Ready := #_w5 AND (#CurrentPUNRdyDly_DInt >= #IN_Configuration.Parameters.CycTime_DataDly);
   IF #PMC_Data.EoC.PUN_Ready AND #IN_Configuration.Features.GM_PN THEN
       #PMC_Data.EoC.PUN_GM_Part_Num := '';
       #PMC_Data.EoC.PUN_GM_Part_Num := #IN_Data.Machining_Assembly.GM_PartNumber;
   END_IF;
   IF #PMC_Data.EoC.PUN_Ready AND #IN_Configuration.Features.Opt_Data THEN
       #PMC_Data.EoC.PUN_Optional_Data := '';
       #PMC_Data.EoC.PUN_Optional_Data := #IN_Data.Machining_Assembly.OptionalData;
   END_IF;
   #_w6 := NOT #PMC_Data.EoC.PUN_Ready AND #FB_OneShot[14];   // falling edge
   #FB_OneShot[14] := #PMC_Data.EoC.PUN_Ready;
   IF #_w6 THEN #Last_PUN_Data := #IN_Data.Machining_Assembly.PUNData; END_IF;
END_REGION

REGION Network 18: Copy Interface Filter Data into DB
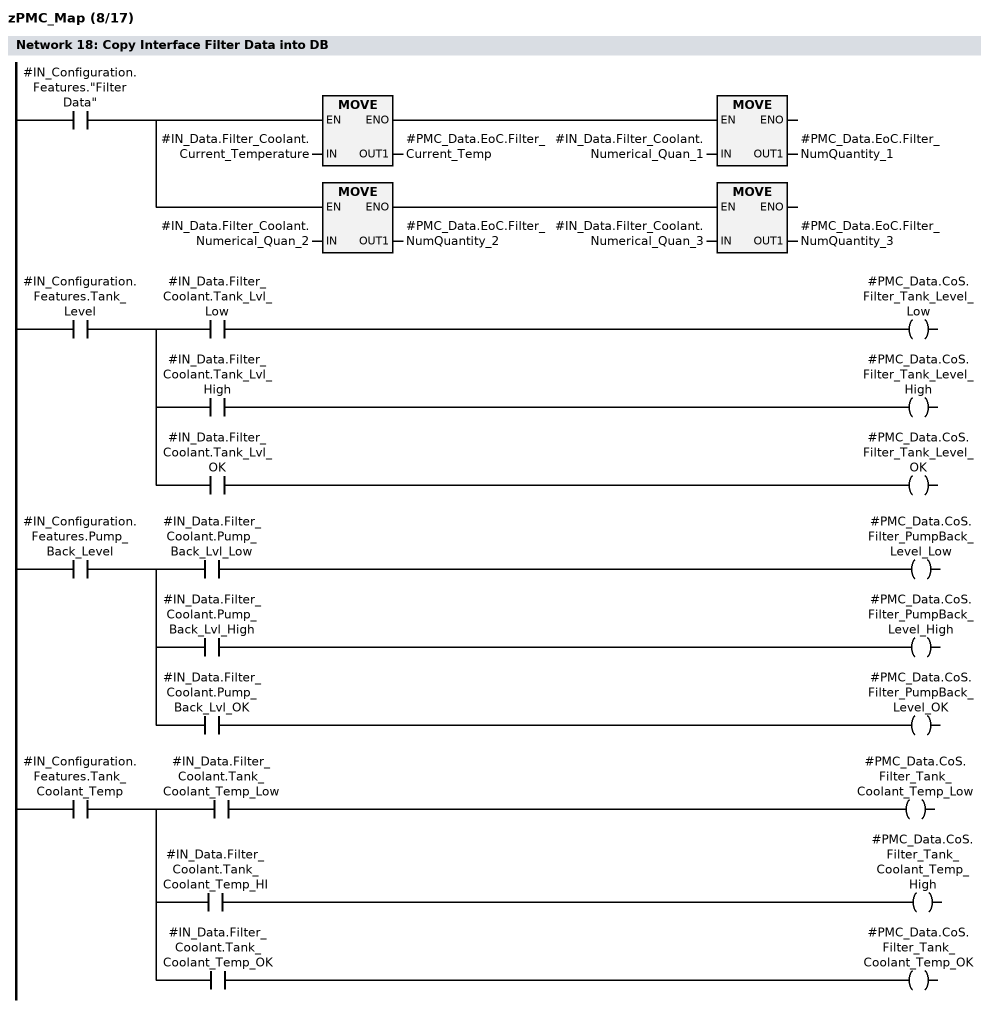
   RUNG wire#powerrail
      Contact( #IN_Configuration.Features."Filter Data" )
      wire#w1
      Move(in := #IN_Data.Filter_Coolant.Current_Temperature, out1 => #PMC_Data.EoC.Filter_Current_Temp)
      Move(in := #IN_Data.Filter_Coolant.Numerical_Quan_1, out1 => #PMC_Data.EoC.Filter_NumQuantity_1)
   END_RUNG
   RUNG wire#w1
      Move(in := #IN_Data.Filter_Coolant.Numerical_Quan_2, out1 => #PMC_Data.EoC.Filter_NumQuantity_2)
      Move(in := #IN_Data.Filter_Coolant.Numerical_Quan_3, out1 => #PMC_Data.EoC.Filter_NumQuantity_3)
   END_RUNG
   RUNG wire#powerrail
      Contact( #IN_Configuration.Features.Tank_Level )
      wire#w2
      Contact( #IN_Data.Filter_Coolant.Tank_Lvl_Low )
      Coil( #PMC_Data.CoS.Filter_Tank_Level_Low )
   END_RUNG
   RUNG wire#w2
      Contact( #IN_Data.Filter_Coolant.Tank_Lvl_High )
      Coil( #PMC_Data.CoS.Filter_Tank_Level_High )
   END_RUNG
   RUNG wire#w2
      Contact( #IN_Data.Filter_Coolant.Tank_Lvl_OK )
      Coil( #PMC_Data.CoS.Filter_Tank_Level_OK )
   END_RUNG
   RUNG wire#powerrail
      Contact( #IN_Configuration.Features.Pump_Back_Level )
      wire#w3
      Contact( #IN_Data.Filter_Coolant.Pump_Back_Lvl_Low )
      Coil( #PMC_Data.CoS.Filter_PumpBack_Level_Low )
   END_RUNG
   RUNG wire#w3
      Contact( #IN_Data.Filter_Coolant.Pump_Back_Lvl_High )
      Coil( #PMC_Data.CoS.Filter_PumpBack_Level_High )
   END_RUNG
   RUNG wire#w3
      Contact( #IN_Data.Filter_Coolant.Pump_Back_Lvl_OK )
      Coil( #PMC_Data.CoS.Filter_PumpBack_Level_OK )
   END_RUNG
   RUNG wire#powerrail
      Contact( #IN_Configuration.Features.Tank_Coolant_Temp )
      wire#w4
      Contact( #IN_Data.Filter_Coolant.Tank_Coolant_Temp_Low )
      Coil( #PMC_Data.CoS.Filter_Tank_Coolant_Temp_Low )
   END_RUNG
   RUNG wire#w4
      Contact( #IN_Data.Filter_Coolant.Tank_Coolant_Temp_HI )
      Coil( #PMC_Data.CoS.Filter_Tank_Coolant_Temp_High )
   END_RUNG
   RUNG wire#w4
      Contact( #IN_Data.Filter_Coolant.Tank_Coolant_Temp_OK )
      Coil( #PMC_Data.CoS.Filter_Tank_Coolant_Temp_OK )
   END_RUNG
   // the same network as SCL:
   IF #IN_Configuration.Features."Filter Data" THEN
       #PMC_Data.EoC.Filter_Current_Temp := #IN_Data.Filter_Coolant.Current_Temperature;
       #PMC_Data.EoC.Filter_NumQuantity_1 := #IN_Data.Filter_Coolant.Numerical_Quan_1;
       #PMC_Data.EoC.Filter_NumQuantity_2 := #IN_Data.Filter_Coolant.Numerical_Quan_2;
       #PMC_Data.EoC.Filter_NumQuantity_3 := #IN_Data.Filter_Coolant.Numerical_Quan_3;
   END_IF;
   #PMC_Data.CoS.Filter_Tank_Level_Low := #IN_Configuration.Features.Tank_Level AND #IN_Data.Filter_Coolant.Tank_Lvl_Low;
   #PMC_Data.CoS.Filter_Tank_Level_High := #IN_Configuration.Features.Tank_Level AND #IN_Data.Filter_Coolant.Tank_Lvl_High;
   #PMC_Data.CoS.Filter_Tank_Level_OK := #IN_Configuration.Features.Tank_Level AND #IN_Data.Filter_Coolant.Tank_Lvl_OK;
   #PMC_Data.CoS.Filter_PumpBack_Level_Low := #IN_Configuration.Features.Pump_Back_Level AND #IN_Data.Filter_Coolant.Pump_Back_Lvl_Low;
   #PMC_Data.CoS.Filter_PumpBack_Level_High := #IN_Configuration.Features.Pump_Back_Level AND #IN_Data.Filter_Coolant.Pump_Back_Lvl_High;
   #PMC_Data.CoS.Filter_PumpBack_Level_OK := #IN_Configuration.Features.Pump_Back_Level AND #IN_Data.Filter_Coolant.Pump_Back_Lvl_OK;
   #PMC_Data.CoS.Filter_Tank_Coolant_Temp_Low := #IN_Configuration.Features.Tank_Coolant_Temp AND #IN_Data.Filter_Coolant.Tank_Coolant_Temp_Low;
   #PMC_Data.CoS.Filter_Tank_Coolant_Temp_High := #IN_Configuration.Features.Tank_Coolant_Temp AND #IN_Data.Filter_Coolant.Tank_Coolant_Temp_HI;
   #PMC_Data.CoS.Filter_Tank_Coolant_Temp_OK := #IN_Configuration.Features.Tank_Coolant_Temp AND #IN_Data.Filter_Coolant.Tank_Coolant_Temp_OK;
END_REGION

REGION Network 19: Copy Interface CMM Data into DB
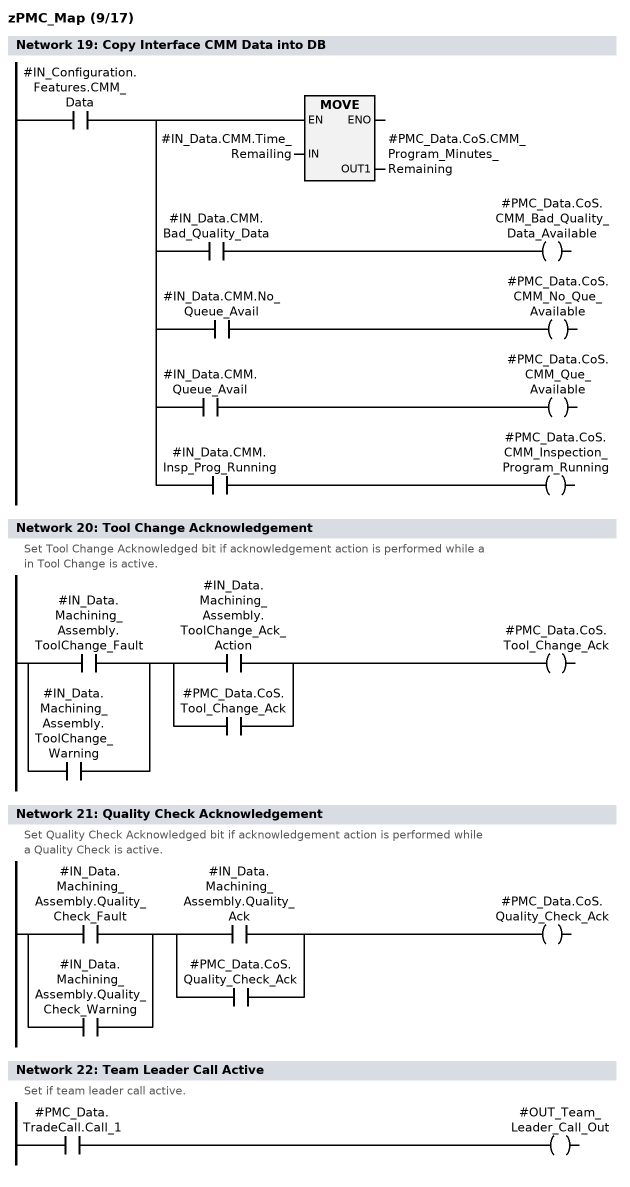
   RUNG wire#powerrail
      Contact( #IN_Configuration.Features.CMM_Data )
      wire#w1
      { S7_GenerateENO := "TRUE" } Move(in := #IN_Data.CMM.Time_Remailing, out1 => #PMC_Data.CoS.CMM_Program_Minutes_Remaining)
   END_RUNG
   RUNG wire#w1
      Contact( #IN_Data.CMM.Bad_Quality_Data )
      Coil( #PMC_Data.CoS.CMM_Bad_Quality_Data_Available )
   END_RUNG
   RUNG wire#w1
      Contact( #IN_Data.CMM.No_Queue_Avail )
      Coil( #PMC_Data.CoS.CMM_No_Que_Available )
   END_RUNG
   RUNG wire#w1
      Contact( #IN_Data.CMM.Queue_Avail )
      Coil( #PMC_Data.CoS.CMM_Que_Available )
   END_RUNG
   RUNG wire#w1
      Contact( #IN_Data.CMM.Insp_Prog_Running )
      Coil( #PMC_Data.CoS.CMM_Inspection_Program_Running )
   END_RUNG
   // the same network as SCL:
   IF #IN_Configuration.Features.CMM_Data THEN
       #PMC_Data.CoS.CMM_Program_Minutes_Remaining := #IN_Data.CMM.Time_Remailing;
   END_IF;
   #PMC_Data.CoS.CMM_Bad_Quality_Data_Available := #IN_Configuration.Features.CMM_Data AND #IN_Data.CMM.Bad_Quality_Data;
   #PMC_Data.CoS.CMM_No_Que_Available := #IN_Configuration.Features.CMM_Data AND #IN_Data.CMM.No_Queue_Avail;
   #PMC_Data.CoS.CMM_Que_Available := #IN_Configuration.Features.CMM_Data AND #IN_Data.CMM.Queue_Avail;
   #PMC_Data.CoS.CMM_Inspection_Program_Running := #IN_Configuration.Features.CMM_Data AND #IN_Data.CMM.Insp_Prog_Running;
END_REGION

REGION Network 20: Tool Change Acknowledgement
   // Set Tool Change Acknowledged bit if acknowledgement action is performed while a 
   // in Tool Change is active.
   RUNG wire#powerrail
      Contact( #IN_Data.Machining_Assembly.ToolChange_Fault )
      wire#w1
      Contact( #IN_Data.Machining_Assembly.ToolChange_Ack_Action )
      wire#w2
      Coil( #PMC_Data.CoS.Tool_Change_Ack )
   END_RUNG
   RUNG wire#powerrail
      Contact( #IN_Data.Machining_Assembly.ToolChange_Warning )
   END_RUNG wire#w1
   RUNG wire#w1
      Contact( #PMC_Data.CoS.Tool_Change_Ack )
   END_RUNG wire#w2
   // the same network as SCL:
   #PMC_Data.CoS.Tool_Change_Ack := (#IN_Data.Machining_Assembly.ToolChange_Fault OR #IN_Data.Machining_Assembly.ToolChange_Warning) AND (#IN_Data.Machining_Assembly.ToolChange_Ack_Action OR #PMC_Data.CoS.Tool_Change_Ack);
END_REGION

REGION Network 21: Quality Check Acknowledgement
   // Set Quality Check Acknowledged bit if acknowledgement action is performed while 
   // a Quality Check is active.
   RUNG wire#powerrail
      Contact( #IN_Data.Machining_Assembly.Quality_Check_Fault )
      wire#w1
      Contact( #IN_Data.Machining_Assembly.Quality_Ack )
      wire#w2
      Coil( #PMC_Data.CoS.Quality_Check_Ack )
   END_RUNG
   RUNG wire#powerrail
      Contact( #IN_Data.Machining_Assembly.Quality_Check_Warning )
   END_RUNG wire#w1
   RUNG wire#w1
      Contact( #PMC_Data.CoS.Quality_Check_Ack )
   END_RUNG wire#w2
   // the same network as SCL:
   #PMC_Data.CoS.Quality_Check_Ack := (#IN_Data.Machining_Assembly.Quality_Check_Fault OR #IN_Data.Machining_Assembly.Quality_Check_Warning) AND (#IN_Data.Machining_Assembly.Quality_Ack OR #PMC_Data.CoS.Quality_Check_Ack);
END_REGION

REGION Network 22: Team Leader Call Active
   // Set if team leader call active.
   RUNG wire#powerrail
      Contact( #PMC_Data.TradeCall.Call_1 )
      Coil( #OUT_Team_Leader_Call_Out )
   END_RUNG
   // the same network as SCL:
   #OUT_Team_Leader_Call_Out := #PMC_Data.TradeCall.Call_1;
END_REGION

REGION Network 23: Counts: Good / Reject / Buffer / Bypass Pallet / Parts Counts: Good and Reject Piece Count
   // When the PM&C Reset bit goes high (from the I.T. system), the PM&C counts are 
   // reset.  Note these counts are monitored by the I.T. system independently from 
   // the production counts that may be maintained separately within the PLC for 
   // other purposes (which is why it is held for an extra scan: to prevent 
   // overwriting by other counters before they are reset)
   // If supplied, the Increment inputs will increment the Piece Count(s) by 
   // P_IncrementAmount for each rising edge.
   // 
   // Additionally, the current cycle time restarts at zero, to prevent cycle time 
   // from last shift from being accumulated (this means that the first cycle will be 
   // shorter than normal in most situations where a cycletime crosses a shift).
   // 
   // Note: Additionally reset of cycletime on shift edge prevents cycletime from 
   // last shift from being accumulated.
   // 
   // The tag BypassPalletOrBufferCnt is used in both Machining 
   // and Assembly Type Maps.  The text Buffer Count is the Machining Side and the Bypass 
   // Pallet Count is the Assembly Side.  There is No Bypass Pallet Count in 
   // Machining and there is No Buffer Count in Assembly.
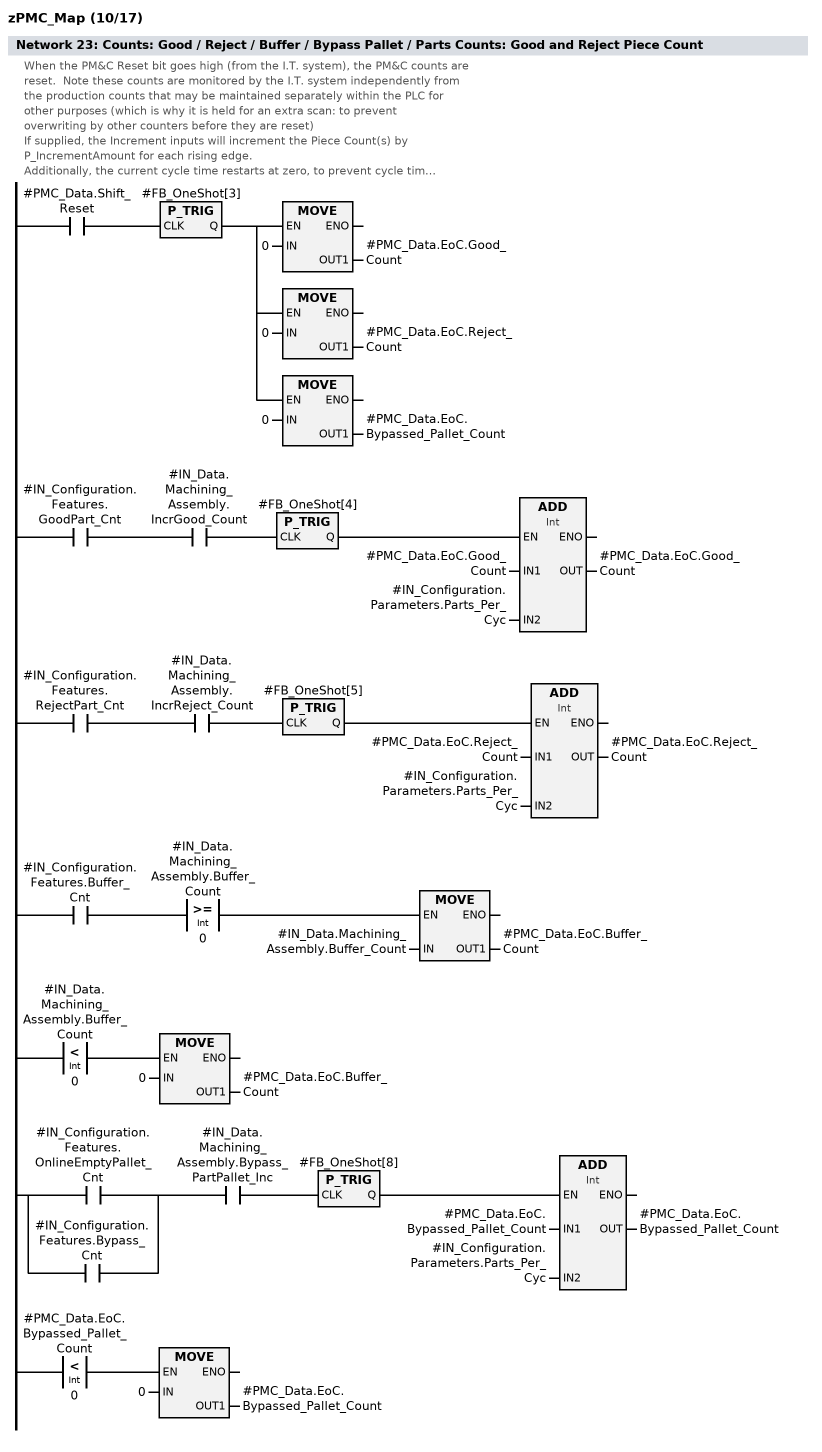
   RUNG wire#powerrail
      Contact( #PMC_Data.Shift_Reset )
      P_Trig( #FB_OneShot[3] )
      wire#w1
      { S7_GenerateENO := "TRUE" } Move(in := 0, out1 => #PMC_Data.EoC.Good_Count)
   END_RUNG
   RUNG wire#w1
      { S7_GenerateENO := "TRUE" } Move(in := 0, out1 => #PMC_Data.EoC.Reject_Count)
   END_RUNG
   RUNG wire#w1
      { S7_GenerateENO := "TRUE" } Move(in := 0, out1 => #PMC_Data.EoC.Bypassed_Pallet_Count)
   END_RUNG
   RUNG wire#powerrail
      Contact( #IN_Configuration.Features.GoodPart_Cnt )
      Contact( #IN_Data.Machining_Assembly.IncrGood_Count )
      P_Trig( #FB_OneShot[4] )
      { S7_Templates := "SrcType := Int"; S7_GenerateENO := "TRUE" } Add(in1 := #PMC_Data.EoC.Good_Count, in2 := #IN_Configuration.Parameters.Parts_Per_Cyc, out => #PMC_Data.EoC.Good_Count)
   END_RUNG
   RUNG wire#powerrail
      Contact( #IN_Configuration.Features.RejectPart_Cnt )
      Contact( #IN_Data.Machining_Assembly.IncrReject_Count )
      P_Trig( #FB_OneShot[5] )
      { S7_Templates := "SrcType := Int"; S7_GenerateENO := "TRUE" } Add(in1 := #PMC_Data.EoC.Reject_Count, in2 := #IN_Configuration.Parameters.Parts_Per_Cyc, out => #PMC_Data.EoC.Reject_Count)
   END_RUNG
   RUNG wire#powerrail
      Contact( #IN_Configuration.Features.Buffer_Cnt )
      { S7_Templates := "SrcType := Int" } GE_Contact(in1 := #IN_Data.Machining_Assembly.Buffer_Count, in2 := 0)
      { S7_GenerateENO := "TRUE" } Move(in := #IN_Data.Machining_Assembly.Buffer_Count, out1 => #PMC_Data.EoC.Buffer_Count)
   END_RUNG
   RUNG wire#powerrail
      { S7_Templates := "SrcType := Int" } LT_Contact(in1 := #IN_Data.Machining_Assembly.Buffer_Count, in2 := 0)
      { S7_GenerateENO := "TRUE" } Move(in := 0, out1 => #PMC_Data.EoC.Buffer_Count)
   END_RUNG
   RUNG wire#powerrail
      Contact( #IN_Configuration.Features.OnlineEmptyPallet_Cnt )
      wire#w2
      Contact( #IN_Data.Machining_Assembly.Bypass_PartPallet_Inc )
      P_Trig( #FB_OneShot[8] )
      { S7_Templates := "SrcType := Int"; S7_GenerateENO := "TRUE" } Add(in1 := #PMC_Data.EoC.Bypassed_Pallet_Count, in2 := #IN_Configuration.Parameters.Parts_Per_Cyc, out => #PMC_Data.EoC.Bypassed_Pallet_Count)
   END_RUNG
   RUNG wire#powerrail
      Contact( #IN_Configuration.Features.Bypass_Cnt )
   END_RUNG wire#w2
   RUNG wire#powerrail
      { S7_Templates := "SrcType := Int" } LT_Contact(in1 := #PMC_Data.EoC.Bypassed_Pallet_Count, in2 := 0)
      { S7_GenerateENO := "TRUE" } Move(in := 0, out1 => #PMC_Data.EoC.Bypassed_Pallet_Count)
   END_RUNG
   // the same network as SCL:
   #_w1 := #PMC_Data.Shift_Reset AND NOT #FB_OneShot[3];   // rising edge
   #FB_OneShot[3] := #PMC_Data.Shift_Reset;
   IF #_w1 THEN
       #PMC_Data.EoC.Good_Count := 0;
       #PMC_Data.EoC.Reject_Count := 0;
       #PMC_Data.EoC.Bypassed_Pallet_Count := 0;
   END_IF;
   #_w2 := #IN_Configuration.Features.GoodPart_Cnt AND #IN_Data.Machining_Assembly.IncrGood_Count;
   #_w3 := #_w2 AND NOT #FB_OneShot[4];   // rising edge
   #FB_OneShot[4] := #_w2;
   IF #_w3 THEN
       #PMC_Data.EoC.Good_Count := #PMC_Data.EoC.Good_Count + #IN_Configuration.Parameters.Parts_Per_Cyc;
   END_IF;
   #_w4 := #IN_Configuration.Features.RejectPart_Cnt AND #IN_Data.Machining_Assembly.IncrReject_Count;
   #_w5 := #_w4 AND NOT #FB_OneShot[5];   // rising edge
   #FB_OneShot[5] := #_w4;
   IF #_w5 THEN
       #PMC_Data.EoC.Reject_Count := #PMC_Data.EoC.Reject_Count + #IN_Configuration.Parameters.Parts_Per_Cyc;
   END_IF;
   IF #IN_Configuration.Features.Buffer_Cnt AND (#IN_Data.Machining_Assembly.Buffer_Count >= 0) THEN
       #PMC_Data.EoC.Buffer_Count := #IN_Data.Machining_Assembly.Buffer_Count;
   END_IF;
   IF #IN_Data.Machining_Assembly.Buffer_Count < 0 THEN #PMC_Data.EoC.Buffer_Count := 0; END_IF;
   #_w6 := (#IN_Configuration.Features.OnlineEmptyPallet_Cnt OR #IN_Configuration.Features.Bypass_Cnt) AND #IN_Data.Machining_Assembly.Bypass_PartPallet_Inc;
   #_w7 := #_w6 AND NOT #FB_OneShot[8];   // rising edge
   #FB_OneShot[8] := #_w6;
   IF #_w7 THEN
       #PMC_Data.EoC.Bypassed_Pallet_Count := #PMC_Data.EoC.Bypassed_Pallet_Count + #IN_Configuration.Parameters.Parts_Per_Cyc;
   END_IF;
   IF #PMC_Data.EoC.Bypassed_Pallet_Count < 0 THEN #PMC_Data.EoC.Bypassed_Pallet_Count := 0; END_IF;
END_REGION

REGION Network 24: Timing: Generate the Cycle End One-shot
   // #Cycle_END_OneShot is a signal which only goes high when the cycle has been 
   // completed, If AutoCycle drops out, and Shift Reset.
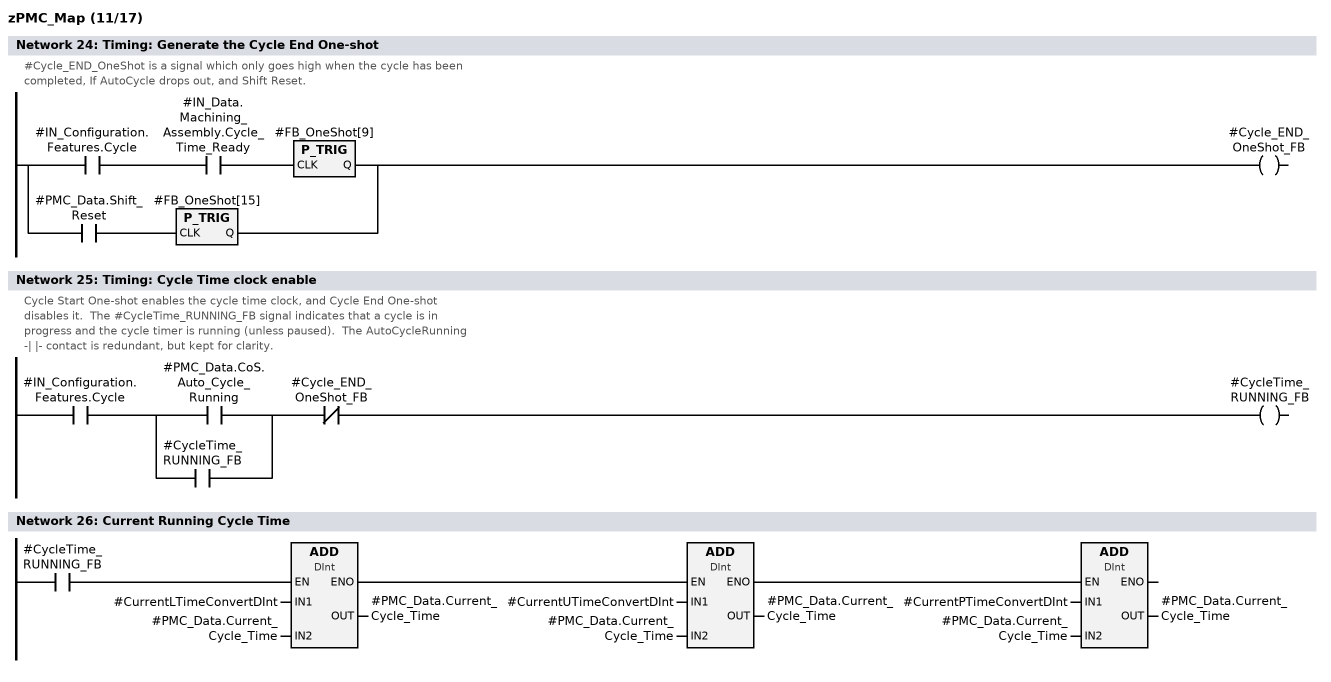
   RUNG wire#powerrail
      Contact( #IN_Configuration.Features.Cycle )
      Contact( #IN_Data.Machining_Assembly.Cycle_Time_Ready )
      P_Trig( #FB_OneShot[9] )
      wire#w1
      Coil( #Cycle_END_OneShot_FB )
   END_RUNG
   RUNG wire#powerrail
      Contact( #PMC_Data.Shift_Reset )
      P_Trig( #FB_OneShot[15] )
   END_RUNG wire#w1
   // the same network as SCL:
   #_w1 := #IN_Configuration.Features.Cycle AND #IN_Data.Machining_Assembly.Cycle_Time_Ready;
   #_w2 := #_w1 AND NOT #FB_OneShot[9];   // rising edge
   #FB_OneShot[9] := #_w1;
   #_w3 := #PMC_Data.Shift_Reset AND NOT #FB_OneShot[15];   // rising edge
   #FB_OneShot[15] := #PMC_Data.Shift_Reset;
   #Cycle_END_OneShot_FB := #_w2 OR #_w3;
END_REGION

REGION Network 25: Timing: Cycle Time clock enable
   // Cycle Start One-shot enables the cycle time clock, and Cycle End One-shot 
   // disables it.  The #CycleTime_RUNNING_FB signal indicates that a cycle is in 
   // progress and the cycle timer is running (unless paused).  The AutoCycleRunning 
   // -| |- contact is redundant, but kept for clarity.
   RUNG wire#powerrail
      Contact( #IN_Configuration.Features.Cycle )
      wire#w1
      Contact( #PMC_Data.CoS.Auto_Cycle_Running )
      wire#w2
      I_Contact( #Cycle_END_OneShot_FB )
      Coil( #CycleTime_RUNNING_FB )
   END_RUNG
   RUNG wire#w1
      Contact( #CycleTime_RUNNING_FB )
   END_RUNG wire#w2
   // the same network as SCL:
   #CycleTime_RUNNING_FB := #IN_Configuration.Features.Cycle AND (#PMC_Data.CoS.Auto_Cycle_Running OR #CycleTime_RUNNING_FB) AND NOT #Cycle_END_OneShot_FB;
END_REGION

REGION Network 26: Current Running Cycle Time
   RUNG wire#powerrail
      Contact( #CycleTime_RUNNING_FB )
      { S7_Templates := "SrcType := DInt" } Add(in1 := #CurrentLTimeConvertDInt, in2 := #PMC_Data.Current_Cycle_Time, out => #PMC_Data.Current_Cycle_Time)
      { S7_Templates := "SrcType := DInt" } Add(in1 := #CurrentUTimeConvertDInt, in2 := #PMC_Data.Current_Cycle_Time, out => #PMC_Data.Current_Cycle_Time)
      { S7_Templates := "SrcType := DInt" } Add(in1 := #CurrentPTimeConvertDInt, in2 := #PMC_Data.Current_Cycle_Time, out => #PMC_Data.Current_Cycle_Time)
   END_RUNG
   // the same network as SCL:
   IF #CycleTime_RUNNING_FB THEN
       #PMC_Data.Current_Cycle_Time := #CurrentLTimeConvertDInt + #PMC_Data.Current_Cycle_Time;
       #PMC_Data.Current_Cycle_Time := #CurrentUTimeConvertDInt + #PMC_Data.Current_Cycle_Time;
       #PMC_Data.Current_Cycle_Time := #CurrentPTimeConvertDInt + #PMC_Data.Current_Cycle_Time;
   END_IF;
END_REGION

REGION Network 27: End of Cycle - Time Transfers / End of Cycle
   // End of cycle duties include moving the current times to the Last Times, and 
   // also setting/resetting other information.
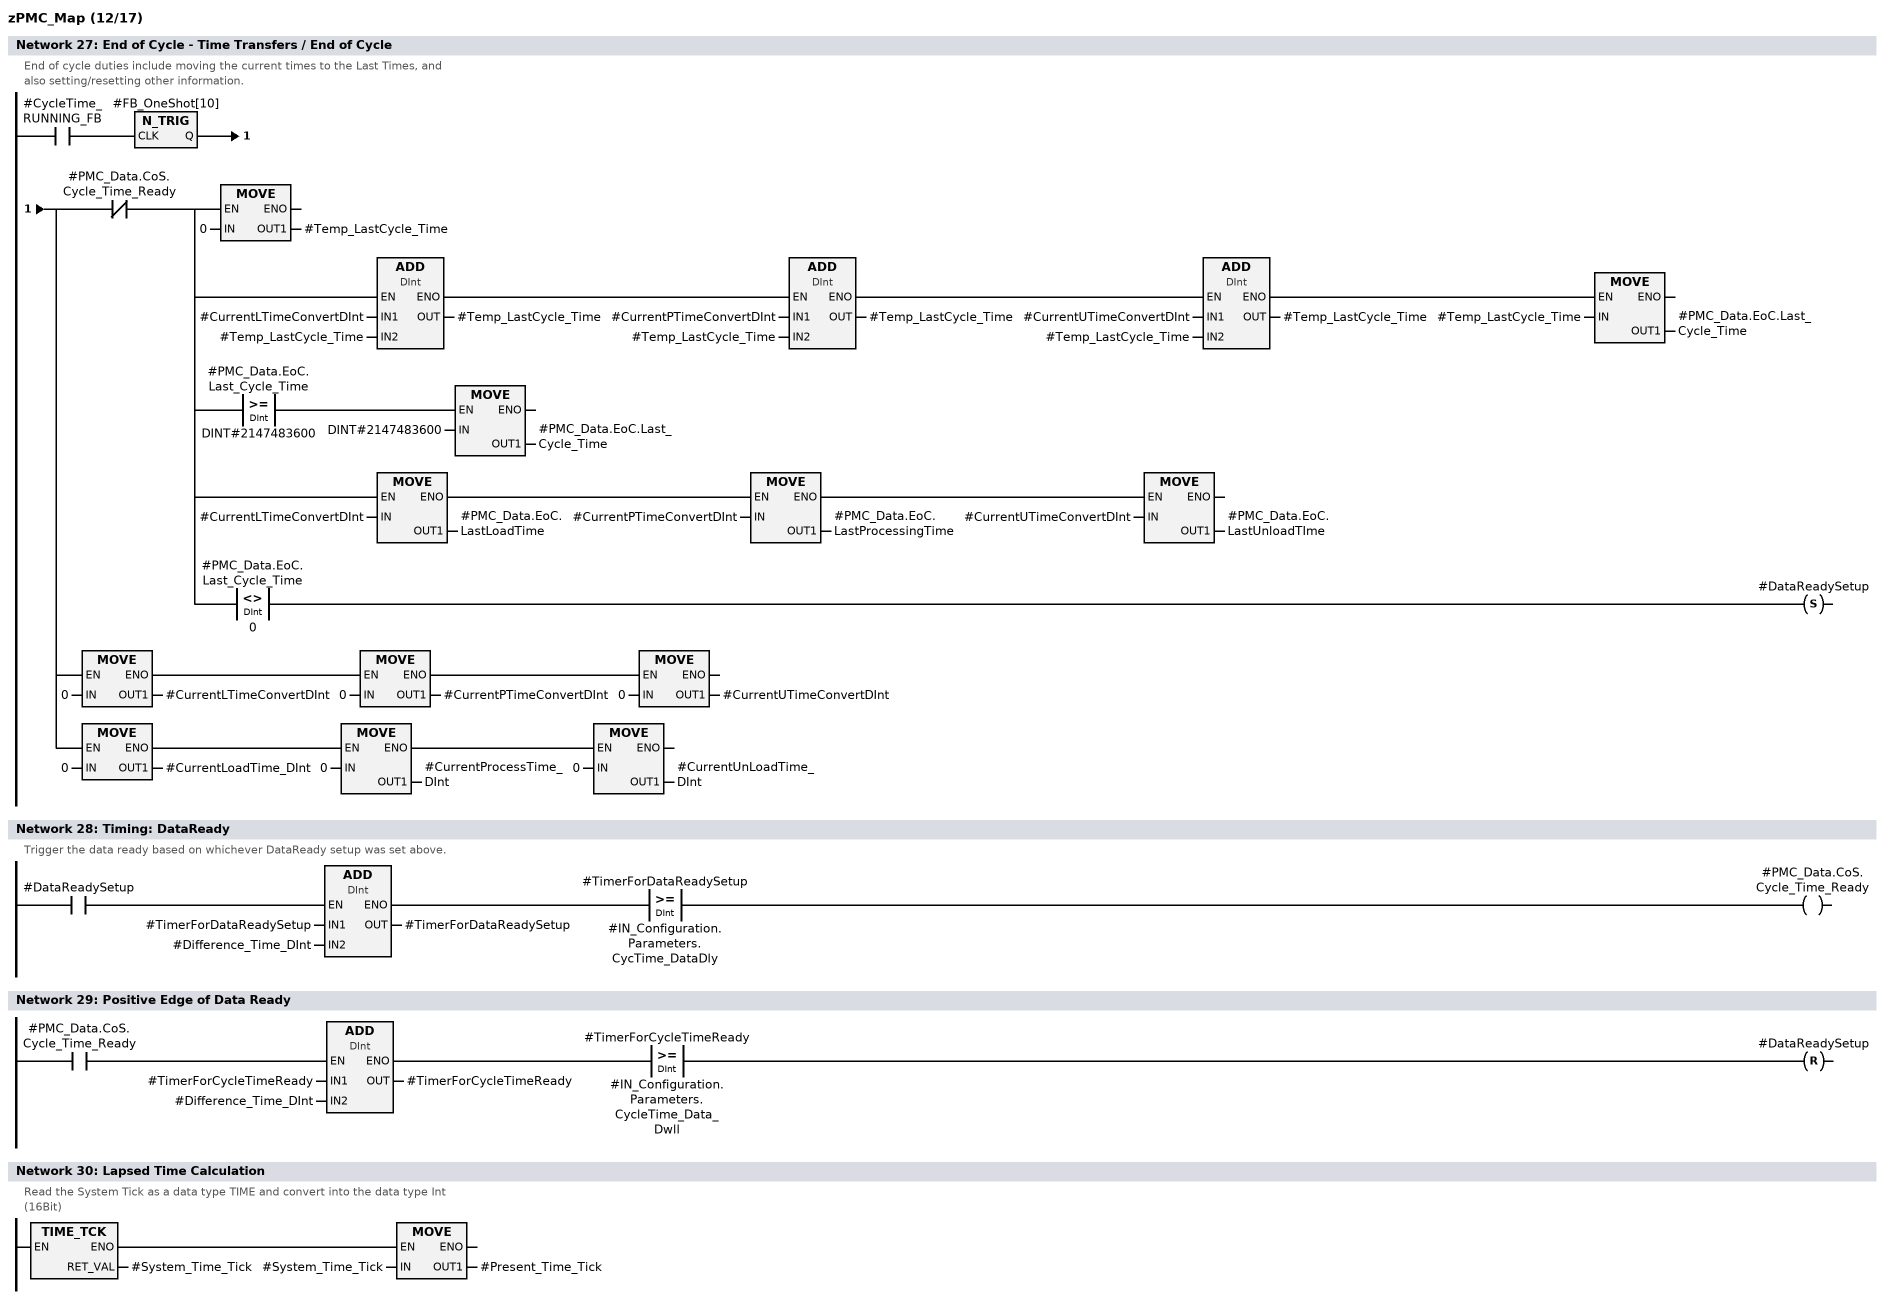
   RUNG wire#powerrail
      Contact( #CycleTime_RUNNING_FB )
      N_Trig( #FB_OneShot[10] )
      wire#w1
      I_Contact( #PMC_Data.CoS.Cycle_Time_Ready )
      wire#w2
      Move(in := 0, out1 => #Temp_LastCycle_Time)
   END_RUNG
   RUNG wire#w2
      { S7_Templates := "SrcType := DInt" } Add(in1 := #CurrentLTimeConvertDInt, in2 := #Temp_LastCycle_Time, out => #Temp_LastCycle_Time)
      { S7_Templates := "SrcType := DInt" } Add(in1 := #CurrentPTimeConvertDInt, in2 := #Temp_LastCycle_Time, out => #Temp_LastCycle_Time)
      { S7_Templates := "SrcType := DInt" } Add(in1 := #CurrentUTimeConvertDInt, in2 := #Temp_LastCycle_Time, out => #Temp_LastCycle_Time)
      Move(in := #Temp_LastCycle_Time, out1 => #PMC_Data.EoC.Last_Cycle_Time)
   END_RUNG
   RUNG wire#w2
      { S7_Templates := "SrcType := DInt" } GE_Contact(in1 := #PMC_Data.EoC.Last_Cycle_Time, in2 := DINT#2147483600)
      Move(in := DINT#2147483600, out1 => #PMC_Data.EoC.Last_Cycle_Time)
   END_RUNG
   RUNG wire#w2
      Move(in := #CurrentLTimeConvertDInt, out1 => #PMC_Data.EoC.LastLoadTime)
      Move(in := #CurrentPTimeConvertDInt, out1 => #PMC_Data.EoC.LastProcessingTime)
      Move(in := #CurrentUTimeConvertDInt, out1 => #PMC_Data.EoC.LastUnloadTIme)
   END_RUNG
   RUNG wire#w2
      { S7_Templates := "SrcType := DInt" } NE_Contact(in1 := #PMC_Data.EoC.Last_Cycle_Time, in2 := 0)
      S_Coil( #DataReadySetup )
   END_RUNG
   RUNG wire#w1
      Move(in := 0, out1 => #CurrentLTimeConvertDInt)
      Move(in := 0, out1 => #CurrentPTimeConvertDInt)
      Move(in := 0, out1 => #CurrentUTimeConvertDInt)
   END_RUNG
   RUNG wire#w1
      Move(in := 0, out1 => #CurrentLoadTime_DInt)
      Move(in := 0, out1 => #CurrentProcessTime_DInt)
      Move(in := 0, out1 => #CurrentUnLoadTime_DInt)
   END_RUNG
   // the same network as SCL:
   #_w1 := NOT #CycleTime_RUNNING_FB AND #FB_OneShot[10];   // falling edge
   #FB_OneShot[10] := #CycleTime_RUNNING_FB;
   #_w2 := #_w1 AND NOT #PMC_Data.CoS.Cycle_Time_Ready;
   IF #_w2 THEN
       #Temp_LastCycle_Time := 0;
       #Temp_LastCycle_Time := #CurrentLTimeConvertDInt + #Temp_LastCycle_Time;
       #Temp_LastCycle_Time := #CurrentPTimeConvertDInt + #Temp_LastCycle_Time;
       #Temp_LastCycle_Time := #CurrentUTimeConvertDInt + #Temp_LastCycle_Time;
       #PMC_Data.EoC.Last_Cycle_Time := #Temp_LastCycle_Time;
   END_IF;
   IF #_w2 AND (#PMC_Data.EoC.Last_Cycle_Time >= DINT#2147483600) THEN
       #PMC_Data.EoC.Last_Cycle_Time := DINT#2147483600;
   END_IF;
   IF #_w2 THEN
       #PMC_Data.EoC.LastLoadTime := #CurrentLTimeConvertDInt;
       #PMC_Data.EoC.LastProcessingTime := #CurrentPTimeConvertDInt;
       #PMC_Data.EoC.LastUnloadTIme := #CurrentUTimeConvertDInt;
   END_IF;
   IF #_w2 AND (#PMC_Data.EoC.Last_Cycle_Time <> 0) THEN #DataReadySetup := TRUE; END_IF;
   IF #_w1 THEN
       #CurrentLTimeConvertDInt := 0;
       #CurrentPTimeConvertDInt := 0;
       #CurrentUTimeConvertDInt := 0;
       #CurrentLoadTime_DInt := 0;
       #CurrentProcessTime_DInt := 0;
       #CurrentUnLoadTime_DInt := 0;
   END_IF;
END_REGION

REGION Network 28: Timing: DataReady
   // Trigger the data ready based on whichever DataReady setup was set above.
   RUNG wire#powerrail
      Contact( #DataReadySetup )
      { S7_Templates := "SrcType := DInt"; S7_GenerateENO := "TRUE" } Add(in1 := #TimerForDataReadySetup, in2 := #Difference_Time_DInt, out => #TimerForDataReadySetup)
      { S7_Templates := "SrcType := DInt" } GE_Contact(in1 := #TimerForDataReadySetup, in2 := #IN_Configuration.Parameters.CycTime_DataDly)
      Coil( #PMC_Data.CoS.Cycle_Time_Ready )
   END_RUNG
   // the same network as SCL:
   // ENO of a box is taken as its EN; it also drops when the box reports an error
   IF #DataReadySetup THEN
       #TimerForDataReadySetup := #TimerForDataReadySetup + #Difference_Time_DInt;
   END_IF;
   #PMC_Data.CoS.Cycle_Time_Ready := #DataReadySetup AND (#TimerForDataReadySetup >= #IN_Configuration.Parameters.CycTime_DataDly);
END_REGION

REGION Network 29: Positive Edge of Data Ready
   RUNG wire#powerrail
      Contact( #PMC_Data.CoS.Cycle_Time_Ready )
      { S7_Templates := "SrcType := DInt"; S7_GenerateENO := "TRUE" } Add(in1 := #TimerForCycleTimeReady, in2 := #Difference_Time_DInt, out => #TimerForCycleTimeReady)
      { S7_Templates := "SrcType := DInt" } GE_Contact(in1 := #TimerForCycleTimeReady, in2 := #IN_Configuration.Parameters.CycleTime_Data_Dwll)
      R_Coil( #DataReadySetup )
   END_RUNG
   // the same network as SCL:
   // ENO of a box is taken as its EN; it also drops when the box reports an error
   IF #PMC_Data.CoS.Cycle_Time_Ready THEN
       #TimerForCycleTimeReady := #TimerForCycleTimeReady + #Difference_Time_DInt;
   END_IF;
   IF #PMC_Data.CoS.Cycle_Time_Ready AND (#TimerForCycleTimeReady >= #IN_Configuration.Parameters.CycleTime_Data_Dwll) THEN
       #DataReadySetup := FALSE;
   END_IF;
END_REGION

REGION Network 30: Lapsed Time Calculation
   // Read the System Tick as a data type TIME and convert into the data type Int 
   // (16Bit)
   RUNG wire#powerrail
      TIME_TCK(RET_VAL => #System_Time_Tick)
      { S7_GenerateENO := "TRUE" } Move(in := #System_Time_Tick, out1 => #Present_Time_Tick)
   END_RUNG
   // the same network as SCL:
   #System_Time_Tick := TIME_TCK(ENO => #_w1);
   IF #_w1 THEN #Present_Time_Tick := #System_Time_Tick; END_IF;
END_REGION

REGION Network 31: Lapsed Time Calculation
   // Calculate time difference beetwen calls in ms
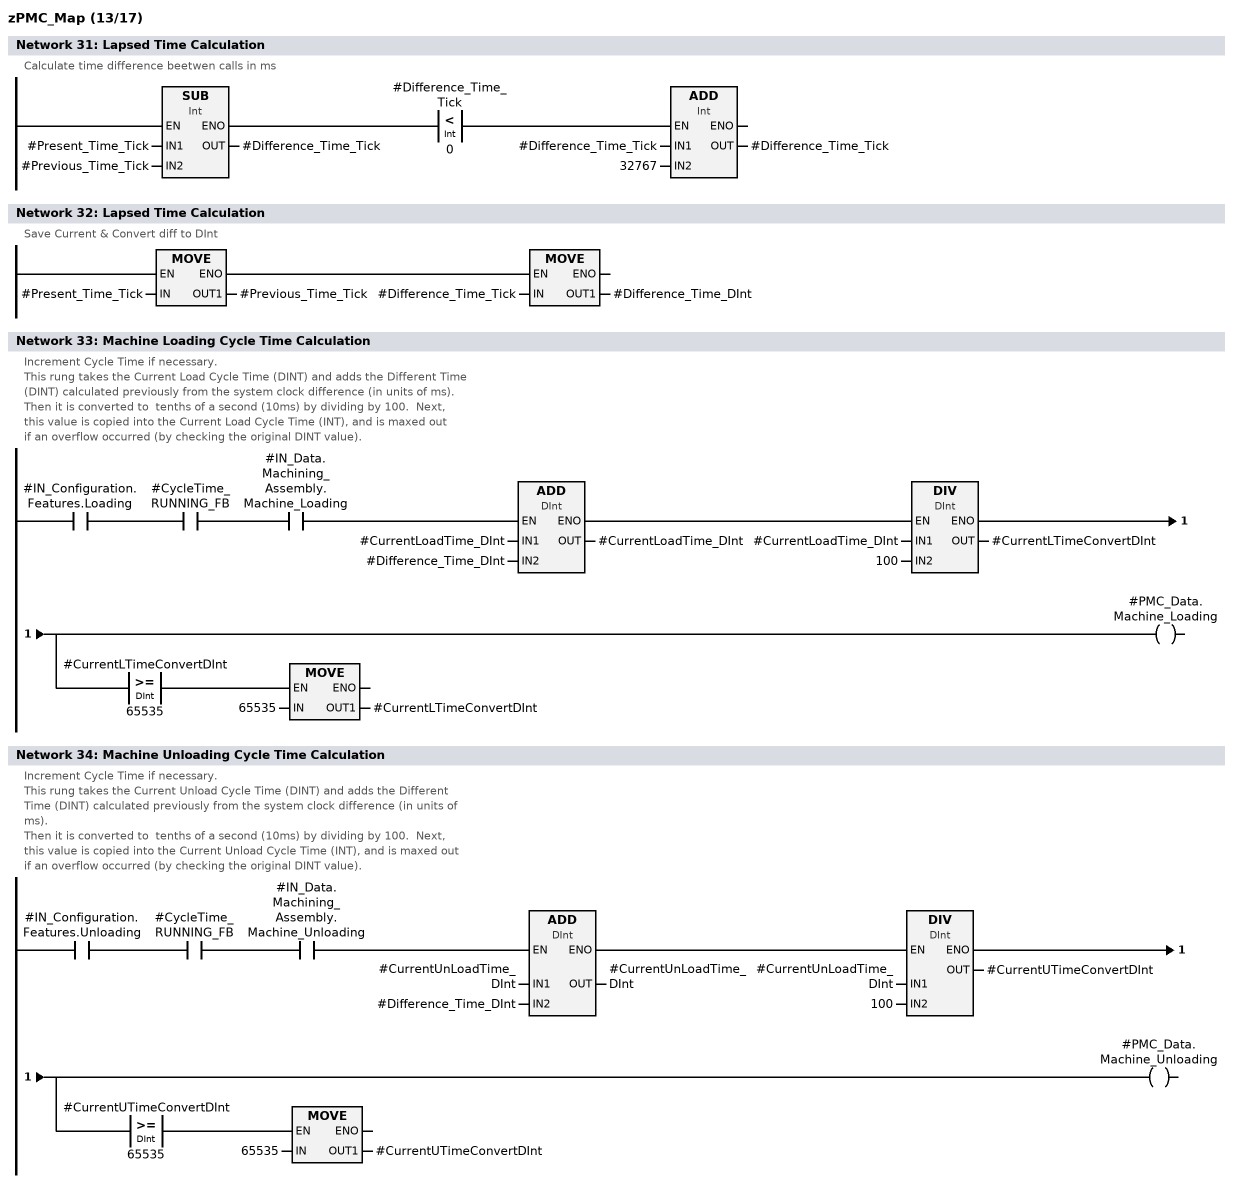
   RUNG wire#powerrail
      { S7_Templates := "SrcType := Int"; S7_GenerateENO := "TRUE" } Sub(in1 := #Present_Time_Tick, in2 := #Previous_Time_Tick, out => #Difference_Time_Tick)
      { S7_Templates := "SrcType := Int" } LT_Contact(in1 := #Difference_Time_Tick, in2 := 0)
      { S7_Templates := "SrcType := Int"; S7_GenerateENO := "TRUE" } Add(in1 := #Difference_Time_Tick, in2 := 32767, out => #Difference_Time_Tick)
   END_RUNG
   // the same network as SCL:
   // ENO of a box is taken as its EN; it also drops when the box reports an error
   #Difference_Time_Tick := #Present_Time_Tick - #Previous_Time_Tick;
   IF #Difference_Time_Tick < 0 THEN #Difference_Time_Tick := #Difference_Time_Tick + 32767; END_IF;
END_REGION

REGION Network 32: Lapsed Time Calculation
   // Save Current & Convert diff to DInt
   RUNG wire#powerrail
      { S7_GenerateENO := "TRUE" } Move(in := #Present_Time_Tick, out1 => #Previous_Time_Tick)
      { S7_GenerateENO := "TRUE" } Move(in := #Difference_Time_Tick, out1 => #Difference_Time_DInt)
   END_RUNG
   // the same network as SCL:
   // ENO of a box is taken as its EN; it also drops when the box reports an error
   #Previous_Time_Tick := #Present_Time_Tick;
   #Difference_Time_DInt := #Difference_Time_Tick;
END_REGION

REGION Network 33: Machine Loading Cycle Time Calculation
   // Increment Cycle Time if necessary.
   // 
   // This rung takes the Current Load Cycle Time (DINT) and adds the Different Time 
   // (DINT) calculated previously from the system clock difference (in units of ms). 
   //  
   // Then it is converted to  tenths of a second (10ms) by dividing by 100.  Next, 
   // this value is copied into the Current Load Cycle Time (INT), and is maxed out 
   // if an overflow occurred (by checking the original DINT value).
   RUNG wire#powerrail
      Contact( #IN_Configuration.Features.Loading )
      Contact( #CycleTime_RUNNING_FB )
      Contact( #IN_Data.Machining_Assembly.Machine_Loading )
      { S7_Templates := "SrcType := DInt"; S7_GenerateENO := "TRUE" } Add(in1 := #CurrentLoadTime_DInt, in2 := #Difference_Time_DInt, out => #CurrentLoadTime_DInt)
      { S7_Templates := "SrcType := DInt"; S7_GenerateENO := "TRUE" } Div(in1 := #CurrentLoadTime_DInt, in2 := 100, out => #CurrentLTimeConvertDInt)
      wire#w1
      Coil( #PMC_Data.Machine_Loading )
   END_RUNG
   RUNG wire#w1
      { S7_Templates := "SrcType := DInt" } GE_Contact(in1 := #CurrentLTimeConvertDInt, in2 := 65535)
      { S7_GenerateENO := "TRUE" } Move(in := 65535, out1 => #CurrentLTimeConvertDInt)
   END_RUNG
   // the same network as SCL:
   // ENO of a box is taken as its EN; it also drops when the box reports an error
   #_w1 := #IN_Configuration.Features.Loading AND #CycleTime_RUNNING_FB AND #IN_Data.Machining_Assembly.Machine_Loading;
   IF #_w1 THEN
       #CurrentLoadTime_DInt := #CurrentLoadTime_DInt + #Difference_Time_DInt;
       #CurrentLTimeConvertDInt := #CurrentLoadTime_DInt / 100;
   END_IF;
   #PMC_Data.Machine_Loading := #_w1;
   IF #_w1 AND (#CurrentLTimeConvertDInt >= 65535) THEN #CurrentLTimeConvertDInt := 65535; END_IF;
END_REGION

REGION Network 34: Machine Unloading Cycle Time Calculation
   // Increment Cycle Time if necessary.
   // 
   // This rung takes the Current Unload Cycle Time (DINT) and adds the Different 
   // Time (DINT) calculated previously from the system clock difference (in units of 
   // ms). 
   //  
   // Then it is converted to  tenths of a second (10ms) by dividing by 100.  Next, 
   // this value is copied into the Current Unload Cycle Time (INT), and is maxed out 
   // if an overflow occurred (by checking the original DINT value).
   RUNG wire#powerrail
      Contact( #IN_Configuration.Features.Unloading )
      Contact( #CycleTime_RUNNING_FB )
      Contact( #IN_Data.Machining_Assembly.Machine_Unloading )
      { S7_Templates := "SrcType := DInt"; S7_GenerateENO := "TRUE" } Add(in1 := #CurrentUnLoadTime_DInt, in2 := #Difference_Time_DInt, out => #CurrentUnLoadTime_DInt)
      { S7_Templates := "SrcType := DInt"; S7_GenerateENO := "TRUE" } Div(in1 := #CurrentUnLoadTime_DInt, in2 := 100, out => #CurrentUTimeConvertDInt)
      wire#w1
      Coil( #PMC_Data.Machine_Unloading )
   END_RUNG
   RUNG wire#w1
      { S7_Templates := "SrcType := DInt" } GE_Contact(in1 := #CurrentUTimeConvertDInt, in2 := 65535)
      { S7_GenerateENO := "TRUE" } Move(in := 65535, out1 => #CurrentUTimeConvertDInt)
   END_RUNG
   // the same network as SCL:
   // ENO of a box is taken as its EN; it also drops when the box reports an error
   #_w1 := #IN_Configuration.Features.Unloading AND #CycleTime_RUNNING_FB AND #IN_Data.Machining_Assembly.Machine_Unloading;
   IF #_w1 THEN
       #CurrentUnLoadTime_DInt := #CurrentUnLoadTime_DInt + #Difference_Time_DInt;
       #CurrentUTimeConvertDInt := #CurrentUnLoadTime_DInt / 100;
   END_IF;
   #PMC_Data.Machine_Unloading := #_w1;
   IF #_w1 AND (#CurrentUTimeConvertDInt >= 65535) THEN #CurrentUTimeConvertDInt := 65535; END_IF;
END_REGION

REGION Network 35: Machine Processing Time Calculation
   // Increment Cycle Time if necessary.
   // 
   // This rung takes the Current Processing Cycle Time (DINT) and adds the Different 
   // Time (DINT) calculated previously from the system clock difference (in units of 
   // ms). 
   //  
   // Then it is converted to  tenths of a second (10ms) by dividing by 100.  Next, 
   // this value is copied into the Current Processing Cycle Time (INT), and is maxed 
   // out if an overflow occurred (by checking the original DINT value).
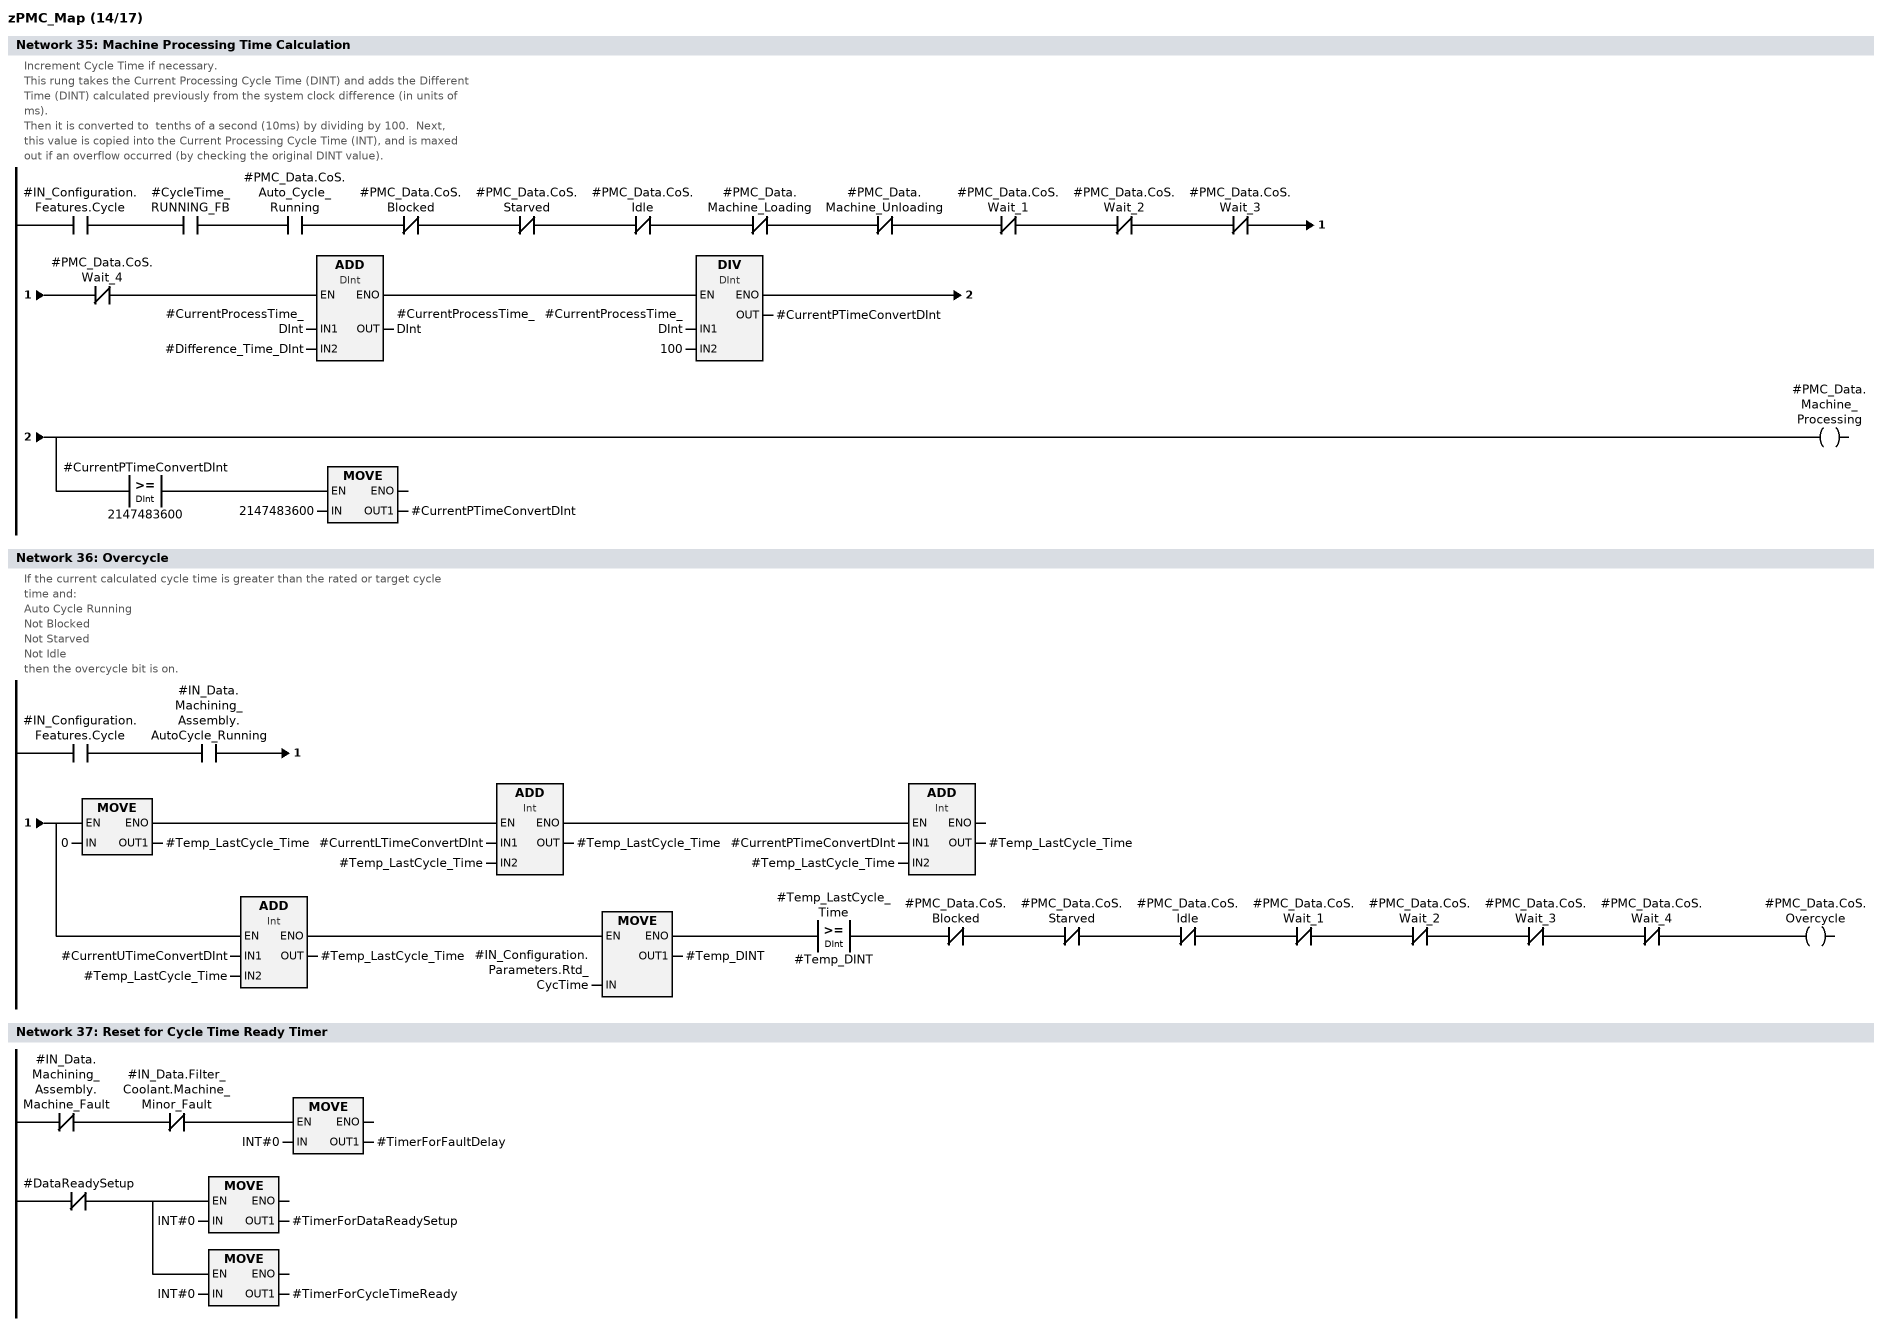
   RUNG wire#powerrail
      Contact( #IN_Configuration.Features.Cycle )
      Contact( #CycleTime_RUNNING_FB )
      Contact( #PMC_Data.CoS.Auto_Cycle_Running )
      I_Contact( #PMC_Data.CoS.Blocked )
      I_Contact( #PMC_Data.CoS.Starved )
      I_Contact( #PMC_Data.CoS.Idle )
      I_Contact( #PMC_Data.Machine_Loading )
      I_Contact( #PMC_Data.Machine_Unloading )
      I_Contact( #PMC_Data.CoS.Wait_1 )
      I_Contact( #PMC_Data.CoS.Wait_2 )
      I_Contact( #PMC_Data.CoS.Wait_3 )
      I_Contact( #PMC_Data.CoS.Wait_4 )
      { S7_Templates := "SrcType := DInt"; S7_GenerateENO := "TRUE" } Add(in1 := #CurrentProcessTime_DInt, in2 := #Difference_Time_DInt, out => #CurrentProcessTime_DInt)
      { S7_Templates := "SrcType := DInt"; S7_GenerateENO := "TRUE" } Div(in1 := #CurrentProcessTime_DInt, in2 := 100, out => #CurrentPTimeConvertDInt)
      wire#w1
      Coil( #PMC_Data.Machine_Processing )
   END_RUNG
   RUNG wire#w1
      { S7_Templates := "SrcType := DInt" } GE_Contact(in1 := #CurrentPTimeConvertDInt, in2 := 2147483600)
      { S7_GenerateENO := "TRUE" } Move(in := 2147483600, out1 => #CurrentPTimeConvertDInt)
   END_RUNG
   // the same network as SCL:
   // ENO of a box is taken as its EN; it also drops when the box reports an error
   #_w1 := #IN_Configuration.Features.Cycle AND #CycleTime_RUNNING_FB AND #PMC_Data.CoS.Auto_Cycle_Running AND NOT #PMC_Data.CoS.Blocked AND NOT #PMC_Data.CoS.Starved AND NOT #PMC_Data.CoS.Idle AND NOT #PMC_Data.Machine_Loading AND NOT #PMC_Data.Machine_Unloading AND NOT #PMC_Data.CoS.Wait_1 AND NOT #PMC_Data.CoS.Wait_2 AND NOT #PMC_Data.CoS.Wait_3 AND NOT #PMC_Data.CoS.Wait_4;
   IF #_w1 THEN
       #CurrentProcessTime_DInt := #CurrentProcessTime_DInt + #Difference_Time_DInt;
       #CurrentPTimeConvertDInt := #CurrentProcessTime_DInt / 100;
   END_IF;
   #PMC_Data.Machine_Processing := #_w1;
   IF #_w1 AND (#CurrentPTimeConvertDInt >= 2147483600) THEN #CurrentPTimeConvertDInt := 2147483600; END_IF;
END_REGION

REGION Network 36: Overcycle
   // If the current calculated cycle time is greater than the rated or target cycle 
   // time and:
   // Auto Cycle Running
   // Not Blocked
   // Not Starved
   // Not Idle
   // then the overcycle bit is on.
   RUNG wire#powerrail
      Contact( #IN_Configuration.Features.Cycle )
      Contact( #IN_Data.Machining_Assembly.AutoCycle_Running )
      wire#w1
      Move(in := 0, out1 => #Temp_LastCycle_Time)
      { S7_Templates := "SrcType := Int" } Add(in1 := #CurrentLTimeConvertDInt, in2 := #Temp_LastCycle_Time, out => #Temp_LastCycle_Time)
      { S7_Templates := "SrcType := Int" } Add(in1 := #CurrentPTimeConvertDInt, in2 := #Temp_LastCycle_Time, out => #Temp_LastCycle_Time)
   END_RUNG
   RUNG wire#w1
      { S7_Templates := "SrcType := Int" } Add(in1 := #CurrentUTimeConvertDInt, in2 := #Temp_LastCycle_Time, out => #Temp_LastCycle_Time)
      Move(in := #IN_Configuration.Parameters.Rtd_CycTime, out1 => #Temp_DINT)
      { S7_Templates := "SrcType := DInt" } GE_Contact(in1 := #Temp_LastCycle_Time, in2 := #Temp_DINT)
      I_Contact( #PMC_Data.CoS.Blocked )
      I_Contact( #PMC_Data.CoS.Starved )
      I_Contact( #PMC_Data.CoS.Idle )
      I_Contact( #PMC_Data.CoS.Wait_1 )
      I_Contact( #PMC_Data.CoS.Wait_2 )
      I_Contact( #PMC_Data.CoS.Wait_3 )
      I_Contact( #PMC_Data.CoS.Wait_4 )
      Coil( #PMC_Data.CoS.Overcycle )
   END_RUNG
   // the same network as SCL:
   #_w1 := #IN_Configuration.Features.Cycle AND #IN_Data.Machining_Assembly.AutoCycle_Running;
   IF #_w1 THEN
       #Temp_LastCycle_Time := 0;
       #Temp_LastCycle_Time := #CurrentLTimeConvertDInt + #Temp_LastCycle_Time;
       #Temp_LastCycle_Time := #CurrentPTimeConvertDInt + #Temp_LastCycle_Time;
       #Temp_LastCycle_Time := #CurrentUTimeConvertDInt + #Temp_LastCycle_Time;
       #Temp_DINT := #IN_Configuration.Parameters.Rtd_CycTime;
   END_IF;
   #PMC_Data.CoS.Overcycle := #_w1 AND (#Temp_LastCycle_Time >= #Temp_DINT) AND NOT #PMC_Data.CoS.Blocked AND NOT #PMC_Data.CoS.Starved AND NOT #PMC_Data.CoS.Idle AND NOT #PMC_Data.CoS.Wait_1 AND NOT #PMC_Data.CoS.Wait_2 AND NOT #PMC_Data.CoS.Wait_3 AND NOT #PMC_Data.CoS.Wait_4;
END_REGION

REGION Network 37: Reset for Cycle Time Ready Timer
   RUNG wire#powerrail
      I_Contact( #IN_Data.Machining_Assembly.Machine_Fault )
      I_Contact( #IN_Data.Filter_Coolant.Machine_Minor_Fault )
      { S7_GenerateENO := "TRUE" } Move(in := INT#0, out1 => #TimerForFaultDelay)
   END_RUNG
   RUNG wire#powerrail
      I_Contact( #DataReadySetup )
      wire#w1
      { S7_GenerateENO := "TRUE" } Move(in := INT#0, out1 => #TimerForDataReadySetup)
   END_RUNG
   RUNG wire#w1
      { S7_GenerateENO := "TRUE" } Move(in := INT#0, out1 => #TimerForCycleTimeReady)
   END_RUNG
   // the same network as SCL:
   IF NOT #IN_Data.Machining_Assembly.Machine_Fault AND NOT #IN_Data.Filter_Coolant.Machine_Minor_Fault THEN
       #TimerForFaultDelay := INT#0;
   END_IF;
   IF NOT #DataReadySetup THEN
       #TimerForDataReadySetup := INT#0;
       #TimerForCycleTimeReady := INT#0;
   END_IF;
END_REGION

REGION Network 38: I.T. Handshake
   // The I.T. system reads this bit to verify that the communication with the 
   // control system is not disrupted. The bit is toggled by the controller between 
   // on and off in 20 second intervals.  This bit should therefore toggle 
   // indefinitely.
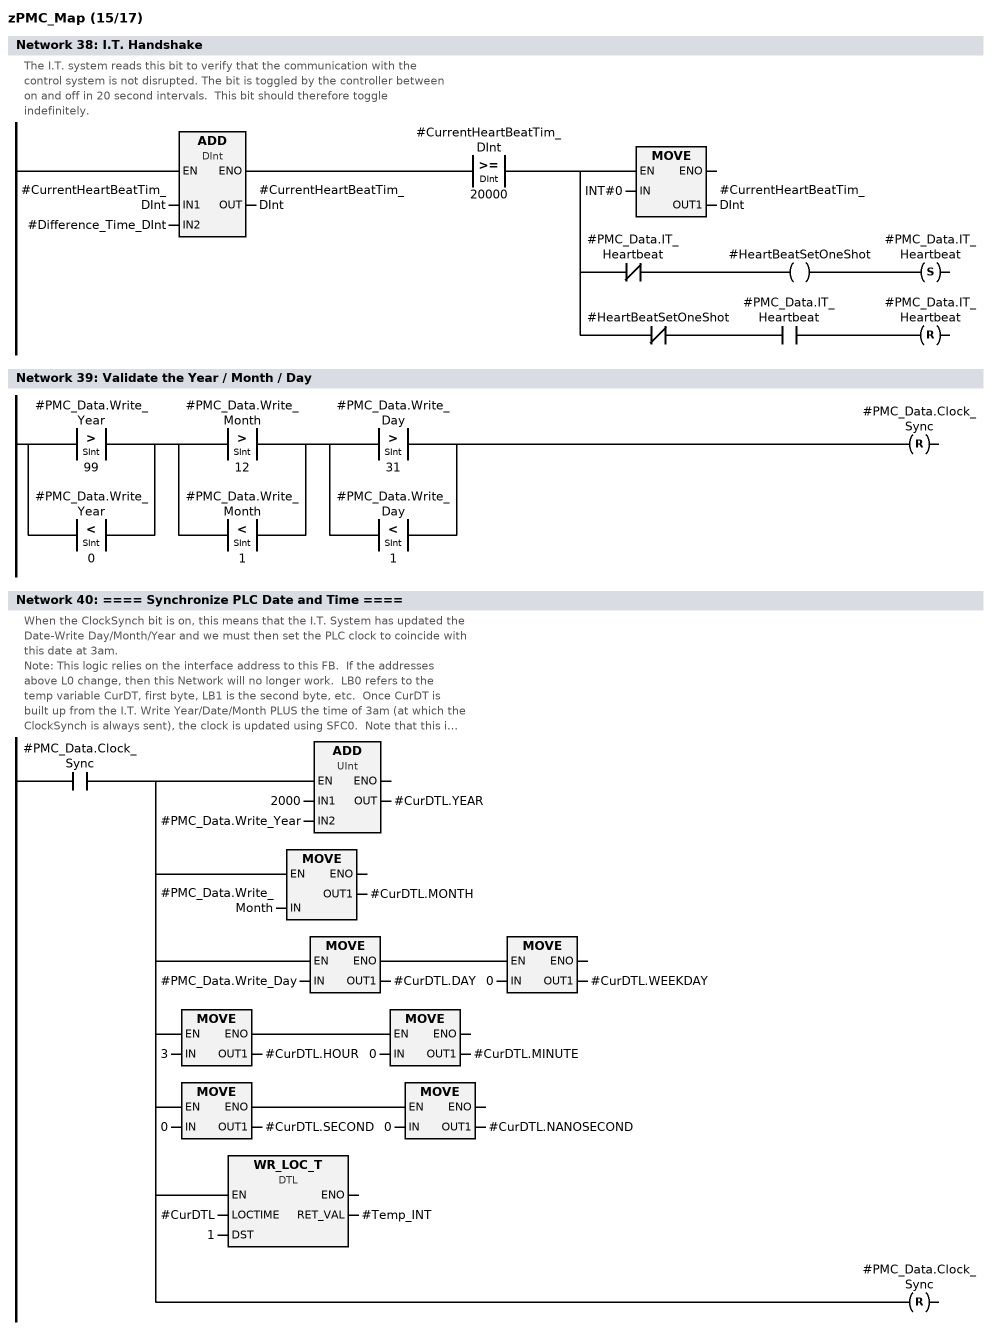
   RUNG wire#powerrail
      { S7_Templates := "SrcType := DInt"; S7_GenerateENO := "TRUE" } Add(in1 := #CurrentHeartBeatTim_DInt, in2 := #Difference_Time_DInt, out => #CurrentHeartBeatTim_DInt)
      { S7_Templates := "SrcType := DInt" } GE_Contact(in1 := #CurrentHeartBeatTim_DInt, in2 := 20000)
      wire#w1
      { S7_GenerateENO := "TRUE" } Move(in := INT#0, out1 => #CurrentHeartBeatTim_DInt)
   END_RUNG
   RUNG wire#w1
      I_Contact( #PMC_Data.IT_Heartbeat )
      Coil( #HeartBeatSetOneShot )
      S_Coil( #PMC_Data.IT_Heartbeat )
   END_RUNG
   RUNG wire#w1
      I_Contact( #HeartBeatSetOneShot )
      Contact( #PMC_Data.IT_Heartbeat )
      R_Coil( #PMC_Data.IT_Heartbeat )
   END_RUNG
   // the same network as SCL:
   // ENO of a box is taken as its EN; it also drops when the box reports an error
   #CurrentHeartBeatTim_DInt := #CurrentHeartBeatTim_DInt + #Difference_Time_DInt;
   #_w1 := #CurrentHeartBeatTim_DInt >= 20000;
   IF #_w1 THEN #CurrentHeartBeatTim_DInt := INT#0; END_IF;
   #HeartBeatSetOneShot := #_w1 AND NOT #PMC_Data.IT_Heartbeat;
   IF #HeartBeatSetOneShot THEN #PMC_Data.IT_Heartbeat := TRUE; END_IF;
   IF #_w1 AND NOT #HeartBeatSetOneShot AND #PMC_Data.IT_Heartbeat THEN
       #PMC_Data.IT_Heartbeat := FALSE;
   END_IF;
END_REGION

REGION Network 39: Validate the Year / Month / Day
   RUNG wire#powerrail
      { S7_Templates := "SrcType := SInt" } GT_Contact(in1 := #PMC_Data.Write_Year, in2 := 99)
      wire#w1
      { S7_Templates := "SrcType := SInt" } GT_Contact(in1 := #PMC_Data.Write_Month, in2 := 12)
      wire#w2
      { S7_Templates := "SrcType := SInt" } GT_Contact(in1 := #PMC_Data.Write_Day, in2 := 31)
      wire#w3
      R_Coil( #PMC_Data.Clock_Sync )
   END_RUNG
   RUNG wire#powerrail
      { S7_Templates := "SrcType := SInt" } LT_Contact(in1 := #PMC_Data.Write_Year, in2 := 0)
   END_RUNG wire#w1
   RUNG wire#w1
      { S7_Templates := "SrcType := SInt" } LT_Contact(in1 := #PMC_Data.Write_Month, in2 := 1)
   END_RUNG wire#w2
   RUNG wire#w2
      { S7_Templates := "SrcType := SInt" } LT_Contact(in1 := #PMC_Data.Write_Day, in2 := 1)
   END_RUNG wire#w3
   // the same network as SCL:
   IF ((#PMC_Data.Write_Year > 99) OR (#PMC_Data.Write_Year < 0)) AND ((#PMC_Data.Write_Month > 12) OR (#PMC_Data.Write_Month < 1)) AND ((#PMC_Data.Write_Day > 31) OR (#PMC_Data.Write_Day < 1)) THEN
       #PMC_Data.Clock_Sync := FALSE;
   END_IF;
END_REGION

REGION Network 40: ==== Synchronize PLC Date and Time ====
   // When the ClockSynch bit is on, this means that the I.T. System has updated the 
   // Date-Write Day/Month/Year and we must then set the PLC clock to coincide with 
   // this date at 3am.
   // 
   // Note: This logic relies on the interface address to this FB.  If the addresses 
   // above L0 change, then this Network will no longer work.  LB0 refers to the 
   // temp variable CurDT, first byte, LB1 is the second byte, etc.  Once CurDT is 
   // built up from the I.T. Write Year/Date/Month PLUS the time of 3am (at which the 
   // ClockSynch is always sent), the clock is updated using SFC0.  Note that this is 
   // independent of the state of the PLC clock before this operation.
   RUNG wire#powerrail
      Contact( #PMC_Data.Clock_Sync )
      wire#w1
      { S7_Templates := "SrcType := UInt" } Add(in1 := 2000, in2 := #PMC_Data.Write_Year, out => #CurDTL.YEAR)
   END_RUNG
   RUNG wire#w1
      { S7_GenerateENO := "TRUE" } Move(in := #PMC_Data.Write_Month, out1 => #CurDTL.MONTH)
   END_RUNG
   RUNG wire#w1
      { S7_GenerateENO := "TRUE" } Move(in := #PMC_Data.Write_Day, out1 => #CurDTL.DAY)
      { S7_GenerateENO := "TRUE" } Move(in := 0, out1 => #CurDTL.WEEKDAY)
   END_RUNG
   RUNG wire#w1
      { S7_GenerateENO := "TRUE" } Move(in := 3, out1 => #CurDTL.HOUR)
      { S7_GenerateENO := "TRUE" } Move(in := 0, out1 => #CurDTL.MINUTE)
   END_RUNG
   RUNG wire#w1
      { S7_GenerateENO := "TRUE" } Move(in := 0, out1 => #CurDTL.SECOND)
      { S7_GenerateENO := "TRUE" } Move(in := 0, out1 => #CurDTL.NANOSECOND)
   END_RUNG
   RUNG wire#w1
      { S7_Templates := "loctime_type := DTL" } WR_LOC_T(LOCTIME := #CurDTL, DST := 1, Ret_Val => #Temp_INT)
   END_RUNG
   RUNG wire#w1
      R_Coil( #PMC_Data.Clock_Sync )
   END_RUNG
   // the same network as SCL:
   // ENO of a box is taken as its EN; it also drops when the box reports an error
   IF #PMC_Data.Clock_Sync THEN
       #CurDTL.YEAR := 2000 + #PMC_Data.Write_Year;
       #CurDTL.MONTH := #PMC_Data.Write_Month;
       #CurDTL.DAY := #PMC_Data.Write_Day;
       #CurDTL.WEEKDAY := 0;
       #CurDTL.HOUR := 3;
       #CurDTL.MINUTE := 0;
       #CurDTL.SECOND := 0;
       #CurDTL.NANOSECOND := 0;
       #Temp_INT := WR_LOC_T(LOCTIME := #CurDTL, DST := 1);
       #PMC_Data.Clock_Sync := FALSE;
   END_IF;
END_REGION

REGION Network 41: FTQ Logic
   // ===========================
   // 07-10-2014 FTQ 3.1: Added to the Standard MM Block.
   // ===========================
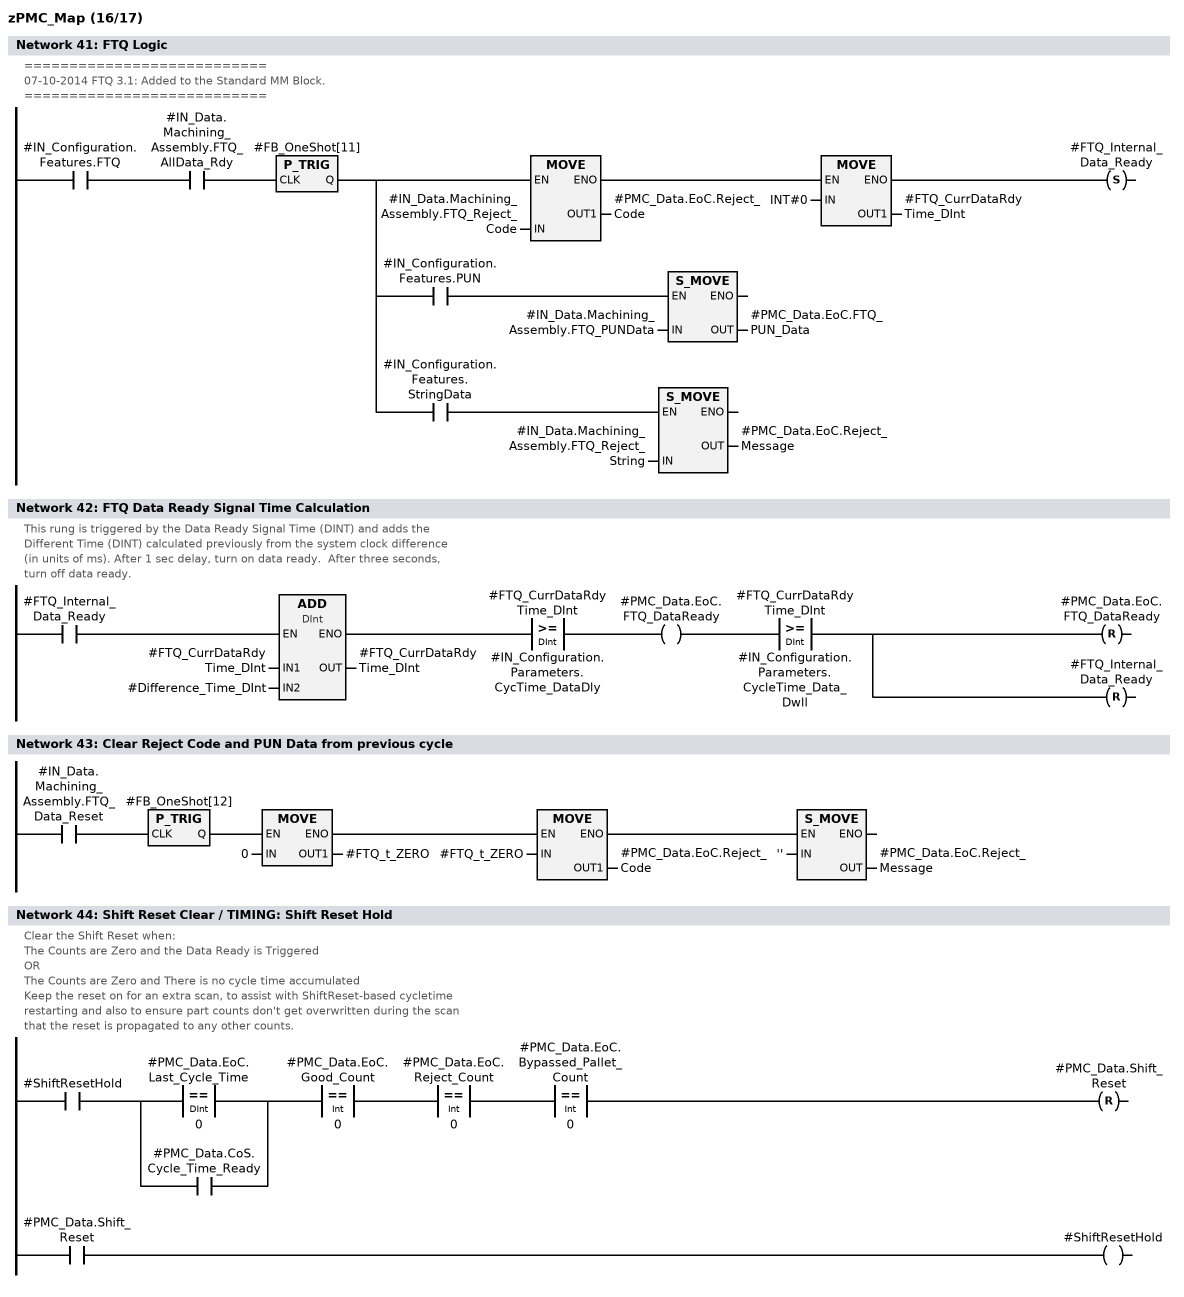
   RUNG wire#powerrail
      Contact( #IN_Configuration.Features.FTQ )
      Contact( #IN_Data.Machining_Assembly.FTQ_AllData_Rdy )
      P_Trig( #FB_OneShot[11] )
      wire#w1
      { S7_GenerateENO := "TRUE" } Move(in := #IN_Data.Machining_Assembly.FTQ_Reject_Code, out1 => #PMC_Data.EoC.Reject_Code)
      { S7_GenerateENO := "TRUE" } Move(in := INT#0, out1 => #FTQ_CurrDataRdyTime_DInt)
      S_Coil( #FTQ_Internal_Data_Ready )
   END_RUNG
   RUNG wire#w1
      Contact( #IN_Configuration.Features.PUN )
      S_Move(in := #IN_Data.Machining_Assembly.FTQ_PUNData, out => #PMC_Data.EoC.FTQ_PUN_Data)
   END_RUNG
   RUNG wire#w1
      Contact( #IN_Configuration.Features.StringData )
      S_Move(in := #IN_Data.Machining_Assembly.FTQ_Reject_String, out => #PMC_Data.EoC.Reject_Message)
   END_RUNG
   // the same network as SCL:
   // ENO of a box is taken as its EN; it also drops when the box reports an error
   #_w1 := #IN_Configuration.Features.FTQ AND #IN_Data.Machining_Assembly.FTQ_AllData_Rdy;
   #_w2 := #_w1 AND NOT #FB_OneShot[11];   // rising edge
   #FB_OneShot[11] := #_w1;
   IF #_w2 THEN
       #PMC_Data.EoC.Reject_Code := #IN_Data.Machining_Assembly.FTQ_Reject_Code;
       #FTQ_CurrDataRdyTime_DInt := INT#0;
       #FTQ_Internal_Data_Ready := TRUE;
   END_IF;
   IF #_w2 AND #IN_Configuration.Features.PUN THEN
       #PMC_Data.EoC.FTQ_PUN_Data := #IN_Data.Machining_Assembly.FTQ_PUNData;
   END_IF;
   IF #_w2 AND #IN_Configuration.Features.StringData THEN
       #PMC_Data.EoC.Reject_Message := #IN_Data.Machining_Assembly.FTQ_Reject_String;
   END_IF;
END_REGION

REGION Network 42: FTQ Data Ready Signal Time Calculation
   // This rung is triggered by the Data Ready Signal Time (DINT) and adds the 
   // Different Time (DINT) calculated previously from the system clock difference 
   // (in units of ms). After 1 sec delay, turn on data ready.  After three seconds, 
   // turn off data ready.
   RUNG wire#powerrail
      Contact( #FTQ_Internal_Data_Ready )
      { S7_Templates := "SrcType := DInt"; S7_GenerateENO := "TRUE" } Add(in1 := #FTQ_CurrDataRdyTime_DInt, in2 := #Difference_Time_DInt, out => #FTQ_CurrDataRdyTime_DInt)
      { S7_Templates := "SrcType := DInt" } GE_Contact(in1 := #FTQ_CurrDataRdyTime_DInt, in2 := #IN_Configuration.Parameters.CycTime_DataDly)
      Coil( #PMC_Data.EoC.FTQ_DataReady )
      { S7_Templates := "SrcType := DInt" } GE_Contact(in1 := #FTQ_CurrDataRdyTime_DInt, in2 := #IN_Configuration.Parameters.CycleTime_Data_Dwll)
      wire#w1
      R_Coil( #PMC_Data.EoC.FTQ_DataReady )
   END_RUNG
   RUNG wire#w1
      R_Coil( #FTQ_Internal_Data_Ready )
   END_RUNG
   // the same network as SCL:
   // ENO of a box is taken as its EN; it also drops when the box reports an error
   IF #FTQ_Internal_Data_Ready THEN
       #FTQ_CurrDataRdyTime_DInt := #FTQ_CurrDataRdyTime_DInt + #Difference_Time_DInt;
   END_IF;
   #PMC_Data.EoC.FTQ_DataReady := #FTQ_Internal_Data_Ready AND (#FTQ_CurrDataRdyTime_DInt >= #IN_Configuration.Parameters.CycTime_DataDly);
   #_w1 := #PMC_Data.EoC.FTQ_DataReady AND (#FTQ_CurrDataRdyTime_DInt >= #IN_Configuration.Parameters.CycleTime_Data_Dwll);
   IF #_w1 THEN
       #PMC_Data.EoC.FTQ_DataReady := FALSE;
       #FTQ_Internal_Data_Ready := FALSE;
   END_IF;
END_REGION

REGION Network 43: Clear Reject Code and PUN Data from previous cycle
   RUNG wire#powerrail
      Contact( #IN_Data.Machining_Assembly.FTQ_Data_Reset )
      P_Trig( #FB_OneShot[12] )
      { S7_GenerateENO := "TRUE" } Move(in := 0, out1 => #FTQ_t_ZERO)
      { S7_GenerateENO := "TRUE" } Move(in := #FTQ_t_ZERO, out1 => #PMC_Data.EoC.Reject_Code)
      S_Move(in := '', out => #PMC_Data.EoC.Reject_Message)
   END_RUNG
   // the same network as SCL:
   // ENO of a box is taken as its EN; it also drops when the box reports an error
   #_w1 := #IN_Data.Machining_Assembly.FTQ_Data_Reset AND NOT #FB_OneShot[12];   // rising edge
   #FB_OneShot[12] := #IN_Data.Machining_Assembly.FTQ_Data_Reset;
   IF #_w1 THEN
       #FTQ_t_ZERO := 0;
       #PMC_Data.EoC.Reject_Code := #FTQ_t_ZERO;
       #PMC_Data.EoC.Reject_Message := '';
   END_IF;
END_REGION

REGION Network 44: Shift Reset Clear / TIMING: Shift Reset Hold
   // Clear the Shift Reset when:
   //      The Counts are Zero and the Data Ready is Triggered
   // OR
   //      The Counts are Zero and There is no cycle time accumulated
   // Keep the reset on for an extra scan, to assist with ShiftReset-based cycletime 
   // restarting and also to ensure part counts don't get overwritten during the scan 
   // that the reset is propagated to any other counts.
   RUNG wire#powerrail
      Contact( #ShiftResetHold )
      wire#w1
      { S7_Templates := "SrcType := DInt" } EQ_Contact(in1 := #PMC_Data.EoC.Last_Cycle_Time, in2 := 0)
      wire#w2
      { S7_Templates := "SrcType := Int" } EQ_Contact(in1 := #PMC_Data.EoC.Good_Count, in2 := 0)
      { S7_Templates := "SrcType := Int" } EQ_Contact(in1 := #PMC_Data.EoC.Reject_Count, in2 := 0)
      { S7_Templates := "SrcType := Int" } EQ_Contact(in1 := #PMC_Data.EoC.Bypassed_Pallet_Count, in2 := 0)
      R_Coil( #PMC_Data.Shift_Reset )
   END_RUNG
   RUNG wire#w1
      Contact( #PMC_Data.CoS.Cycle_Time_Ready )
   END_RUNG wire#w2
   RUNG wire#powerrail
      Contact( #PMC_Data.Shift_Reset )
      Coil( #ShiftResetHold )
   END_RUNG
   // the same network as SCL:
   IF #ShiftResetHold AND ((#PMC_Data.EoC.Last_Cycle_Time = 0) OR #PMC_Data.CoS.Cycle_Time_Ready) AND (#PMC_Data.EoC.Good_Count = 0) AND (#PMC_Data.EoC.Reject_Count = 0) AND (#PMC_Data.EoC.Bypassed_Pallet_Count = 0) THEN
       #PMC_Data.Shift_Reset := FALSE;
   END_IF;
   #ShiftResetHold := #PMC_Data.Shift_Reset;
END_REGION

REGION Network 45: Clear Cycle Timers if Cycle, Load, or Unload are not used
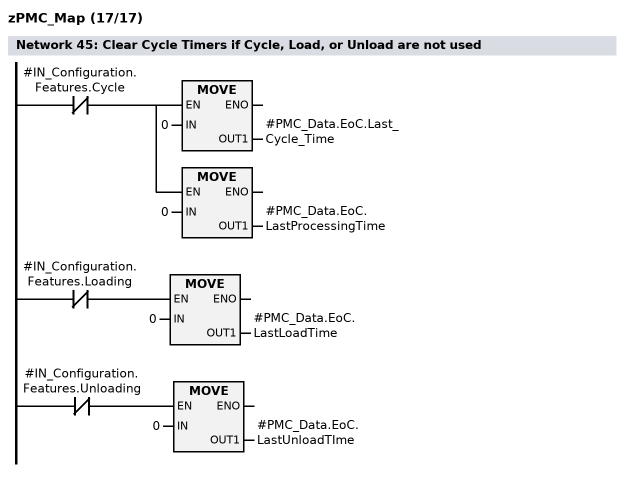
   RUNG wire#powerrail
      I_Contact( #IN_Configuration.Features.Cycle )
      wire#w1
      Move(in := 0, out1 => #PMC_Data.EoC.Last_Cycle_Time)
   END_RUNG
   RUNG wire#w1
      Move(in := 0, out1 => #PMC_Data.EoC.LastProcessingTime)
   END_RUNG
   RUNG wire#powerrail
      I_Contact( #IN_Configuration.Features.Loading )
      Move(in := 0, out1 => #PMC_Data.EoC.LastLoadTime)
   END_RUNG
   RUNG wire#powerrail
      I_Contact( #IN_Configuration.Features.Unloading )
      Move(in := 0, out1 => #PMC_Data.EoC.LastUnloadTIme)
   END_RUNG
   // the same network as SCL:
   IF NOT #IN_Configuration.Features.Cycle THEN
       #PMC_Data.EoC.Last_Cycle_Time := 0;
       #PMC_Data.EoC.LastProcessingTime := 0;
   END_IF;
   IF NOT #IN_Configuration.Features.Loading THEN #PMC_Data.EoC.LastLoadTime := 0; END_IF;
   IF NOT #IN_Configuration.Features.Unloading THEN #PMC_Data.EoC.LastUnloadTIme := 0; END_IF;
END_REGION
END_FUNCTION_BLOCK
